    //==========================================================
    // 21 — WAIT HOMING COMPLETE
    //==========================================================
    21:
        // Start infeed/outfeed only after homing is complete
//        IF lowerKnifeStatusW1.homingComplete THEN
            lowerKnifeInFeedRun  := TRUE;
            lowerKnifeOutFeedRun := TRUE;
            lowerKnifeStep := 40;
//        END_IF

    //==========================================================
    // 40 — NORMAL OPERATION
    //==========================================================
    40:
	
        lowerKnifeJogFw       := lowerKnifeJogFwCmd;
        lowerKnifeJogRev      := lowerKnifeJogRevCmd;	
	
		instTOF_LowerKnifePaperSensor(IN := lowerKnifePaperSensor, PT:= T#30M);	
	
		IF instTOF_LowerKnifePaperSensor.Q  OR lineSpeedMPM > 5 THEN
			
			lowerKnifeInFeedDriveRef := LIMIT(machineConfigLowerKnife.minLineSpeed,
											  lineSpeedMPMRamp,
											  lowerLevelInfeedSpeedLimit) * machineConfigLowerKnife.infeedRollSpeedOffset;
		 
			lowerKnifeOutFeedDriveRef := LIMIT(machineConfigLowerKnife.minLineSpeed,
											   lineSpeedMPMRamp,
											   999) * machineConfigLowerKnife.outfeedRollSpeedOffset;		
		ELSE
			
			lowerKnifeInFeedDriveRef := 0;
			lowerKnifeOutFeedDriveRef := 0;		
			
		END_IF



        // Enable cut only when commanded and paper present
        lowerKnifeCut := (lowerKnifeCutCmd AND lowerKnifePaperSensor);
		
		
		IF NOT measuringWheelPaperPresence THEN
			
			lowerLevelInfeedSpeedLimit := lowerKnifeMaximumSpeedActive;
			
		ELSE
		
			lowerLevelInfeedSpeedLimit := 999;	
		
		END_IF				
		

END_CASE

//==============================================================
// 5) GLOBAL INTERLOCK — IMMEDIATE STOP
//==============================================================
// Immediate stop on any of these conditions:
// - Safety chain not OK
// - Any drive not OK
// - Power OFF command rising edge
IF (NOT safetyFeedback)
   OR (NOT lowerKnifeAllDrivesOK)
   OR lowerKnifeRtPowerOff.Q THEN

    lowerKnifeStep := 0;

    lowerKnifeEnable      := FALSE;
    lowerKnifeSlave1Run   := FALSE;
    lowerKnifeSlave2Run   := FALSE;
    lowerKnifeInFeedRun   := FALSE;
    lowerKnifeOutFeedRun  := FALSE;

    lowerKnifeJogFw       := FALSE;
    lowerKnifeJogRev      := FALSE;
    lowerKnifeHome        := FALSE;
    lowerKnifeCut         := FALSE;

    lowerKnifeInFeedDriveRef  := 0.0;
    lowerKnifeOutFeedDriveRef := 0.0;

    // Reset internal timers for a clean restart
    lowerKnifeTimerWait(IN := FALSE);
    lowerKnifeTimerPulse(IN := FALSE);
    lowerKnifeTimerClear(IN := FALSE);
    lowerKnifeTimerReset(IN := FALSE);
END_IF

//Start Lubrification pump
lowerKnifeLubrification := lowerKnifeEnable;
 


//==============================================================
// ENCODER SELECTION — LOWER KNIFE
//==============================================================
// Copied 1:1 from the provided upper-knife reference logic.
// NOTE: The TRUE/FALSE meaning of "*EncoderSwitch" should match your IO mapping.
//==============================================================


   //----------------------------------------------------------
    // AUTO MODE
    //----------------------------------------------------------
    IF NOT measuringWheelPaperPresence THEN
        // No paper → immediate fallback to measuring wheel encoder
        lowerKnifeEncoderSwitch := TRUE;

        // Reset delay timer
        instTONLowerKnifeSwitchEncoderDelay.IN := FALSE;

    ELSE
        // Paper present → start delay before switching
        instTONLowerKnifeSwitchEncoderDelay.IN := TRUE;

        // Switch only after delay elapsed
        IF instTONLowerKnifeSwitchEncoderDelay.Q THEN
				
			lowerKnifeEncoderSwitch := FALSE;

        END_IF
		
    END_IF

//--------------------------------------------------------------
// TIMER EXECUTION (ALWAYS CALLED)
//--------------------------------------------------------------
instTONLowerKnifeSwitchEncoderDelay(
    PT := machineConfigLowerKnife.switchEncoderDelay
);
END_METHOD

METHOD _03_LineSpeedLimit
VAR_INPUT
END_VAR
//==============================================================
// SHEET LENGTH SELECTION — UPPER / LOWER KNIFE
//==============================================================

CASE currentOrder.levelSelector OF

    //----------------------------------------------------------
    // ORDER 1 ONLY
    //----------------------------------------------------------
    E_LevelSelector.eUpperOnly:
         instFB_SpeedLimitUpperKnife.sheetLength := currentOrder.order1.sheetLength;
		instFB_SpeedLimitLowerKnife.sheetLength := currentOrder.order1.sheetLength;
	 
		instFB_SpeedLimitUpperKnife.knifeEnabled := TRUE;
		instFB_SpeedLimitLowerKnife.knifeEnabled := FALSE;	
    //----------------------------------------------------------
    // ORDER 2 ONLY
    //----------------------------------------------------------
    E_LevelSelector.eLowerOnly:
        instFB_SpeedLimitLowerKnife.sheetLength := currentOrder.order1.sheetLength;
			instFB_SpeedLimitLowerKnife.sheetLength := currentOrder.order1.sheetLength;
	
		instFB_SpeedLimitUpperKnife.knifeEnabled := FALSE;
		instFB_SpeedLimitLowerKnife.knifeEnabled := TRUE;		

    //----------------------------------------------------------
    // BOTH ORDERS
    //----------------------------------------------------------
    E_LevelSelector.eBoth:

		// Inverted mapping
		instFB_SpeedLimitUpperKnife.sheetLength := currentOrder.order1.sheetLength;
		instFB_SpeedLimitLowerKnife.sheetLength := currentOrder.order2.sheetLength;
		instFB_SpeedLimitUpperKnife.knifeEnabled := TRUE;
		instFB_SpeedLimitLowerKnife.knifeEnabled := TRUE;
		

END_CASE

//==============================================================
// UPPER KNIFE — SPEED LIMIT CALCULATION
//==============================================================
instFB_SpeedLimitUpperKnife(
    machineSpeed             := lineSpeedMPM,
    numberOfPoints           := 10,
    machineConfigRotaryKnife := machineConfigUpperKnife,

    reduceLineSpeed          => upperKnifeReduceLineSpeed,
    speedLimitAcive          => upperKnifeSpeedLimit,
    speedCurveActive         => upperKnifeSpeedCurveActive,
    maximumSpeedActive       => upperKnifeMaximumSpeedActive
);

//==============================================================
// LOWER KNIFE — SPEED LIMIT CALCULATION
//==============================================================
instFB_SpeedLimitLowerKnife(
    machineSpeed             := lineSpeedMPM,
    numberOfPoints           := 10,
    machineConfigRotaryKnife := machineConfigLowerKnife,

    reduceLineSpeed          => lowerKnifeReduceLineSpeed,
    speedLimitAcive          => lowerKnifeSpeedLimit,
    speedCurveActive         => lowerKnifeSpeedCurveActive,
    maximumSpeedActive       => lowerKnifeMaximumSpeedActive
);
END_METHOD

METHOD _04_AuxControls
VAR_INPUT
END_VAR

//Start outfeed conveyor
startOutfeedConveyor := upperKnifeEnable OR lowerKnifeEnable;
END_METHOD

METHOD _05_DisplayVariables
VAR_INPUT
END_VAR
(*

    upperKnifeHmiStatus                       : hmiStatus_TypeStruct;
    lowerKnifeHmiStatus                       : hmiStatus_TypeStruct;

    reduceLineSpeed          => upperKnifeReduceLineSpeed,
    speedLimitAcive          => upperKnifeSpeedLimit,
    speedCurveActive         => upperKnifeSpeedCurveActive,
    maximumSpeedActive       => upperKnifeMaximumSpeedActive
	
    upperKnifeStatusW1              : rotaryKnifeStatusWord1_TypeStruct;
    upperKnifeStatusW2              : rotaryKnifeStatusWord2_TypeStruct;
rotaryKnifeStatusWord1_TypeStruct
rotaryKnifeStatusWord1_TypeStruct
    lowerKnifeStatusWord1           : INT;
    lowerKnifeStatusWord2           : INT;
    lowerKnifeModbusDword           : DWORD;
    lowerKnifeWriteMenu2029         : DWORD;
    lowerKnifeLineSpeed             : WORD;
    lowerKnifeStatusW1              : rotaryKnifeStatusWord1_TypeStruct;
    lowerKnifeStatusW2              : rotaryKnifeStatusWord2_TypeStruct;	
	
	
*)
//────────────────────────────────────────────
// LINE SPEED PROCESSING
//────────────────────────────────────────────
IF lineSpeedMPM > 0 THEN
    lineSpeed := TRUNC(lineSpeedMPM);
ELSE
    lineSpeed := 0;
END_IF

//────────────────────────────────────────────
// UPPER KNIFE - STATUS MAPPING
//────────────────────────────────────────────
upperKnifeHmiStatus.maxSpeed         := upperKnifeMaximumSpeedActive;       // Current active maximum speed
upperKnifeHmiStatus.speedLimitActive := upperKnifeSpeedLimit;                // Speed limit status
upperKnifeHmiStatus.speedCurveActive := upperKnifeSpeedCurveActive;

upperKnifeHmiStatus.statusWord1      := upperKnifeStatusW1;                 // General status word 1
upperKnifeHmiStatus.statusWord2      := upperKnifeStatusW2;                 // General status word 2
upperKnifeHmiStatus.totalOfCuts      := upperKnifeTotalOfCutsAccumulator;   // Cumulative cut counter
//────────────────────────────────────────────
// LOWER KNIFE - STATUS MAPPING
//────────────────────────────────────────────
lowerKnifeHmiStatus.maxSpeed         := lowerKnifeMaximumSpeedActive;       // Current active maximum speed
lowerKnifeHmiStatus.speedLimitActive := lowerKnifeSpeedLimit;                // Speed limit status
lowerKnifeHmiStatus.speedCurveActive := lowerKnifeSpeedCurveActive;

lowerKnifeHmiStatus.statusWord1      := lowerKnifeStatusW1;                 // General status word 1
lowerKnifeHmiStatus.statusWord2      := lowerKnifeStatusW2;                 // General status word 2
lowerKnifeHmiStatus.totalOfCuts      := lowerKnifeTotalOfCutsAccumulator;   // Cumulative cut counter
END_METHOD

METHOD _06_TotalOfCuts
VAR_INPUT
END_VAR
// ==========================================================
// UPPER KNIFE CUT DETECTION & COUNTER LOGIC
// ==========================================================

(* Detect rising edge of the upper knife sensor to increment the cut counter *)
IF upperKnifeHomeSensor AND NOT upperKnifeHomeSensorOld THEN
	
	// Increment the cumulative cut count for the upper knife
	upperKnifeTotalOfCutsAccumulator := upperKnifeTotalOfCutsAccumulator + 1;

END_IF

// Store current sensor state for next scan cycle edge detection
upperKnifeHomeSensorOld := upperKnifeHomeSensor;

(* Reset Logic: Clears the upper knife cut counter *)
IF upperKnifeReset THEN
	
	upperKnifeTotalOfCutsAccumulator := 0;

END_IF


// ==========================================================
// LOWER KNIFE CUT DETECTION & COUNTER LOGIC
// ==========================================================

(* Detect rising edge of the lower knife sensor to increment the cut counter *)
IF lowerKnifeHomeSensor AND NOT lowerKnifeHomeSensorOld THEN
	
	// Increment the cumulative cut count for the lower knife
	lowerKnifeTotalOfCutsAccumulator := lowerKnifeTotalOfCutsAccumulator + 1;

END_IF

// Store current sensor state for next scan cycle edge detection
lowerKnifeHomeSensorOld := lowerKnifeHomeSensor;

(* Reset Logic: Clears the lower knife cut counter *)
IF lowerKnifeReset THEN
	
	lowerKnifeTotalOfCutsAccumulator := 0;

END_IF
END_METHOD

METHOD _07_LineSpeedRamp
VAR
	
	rampTargetMPM : REAL;

END_VAR
(*

    lineSpeedMPM                    : REAL;
    aocSpeedMPM                     : REAL;
*)
IF NOT aocRunning THEN
	
	rampTargetMPM := lineSpeedMPM;

ELSE
	
	rampTargetMPM := aocSpeedMPM;

END_IF



// Ramp function block execution
instFB_Gen_SRamp(
    X          := rampTargetMPM,
    A_UP       := 5,
    A_DN       := -5,
    VU_MAX     := 1000.0,
    VD_MAX     := -1000.0,
    LIMIT_HIGH := 350,
	Y => lineSpeedMPMRamp
);




lineSpeedStacker := upperKnifeInFeedDriveRef;
END_METHOD

METHOD _08_StopTheLineCommand
VAR_INPUT
END_VAR

// ======================================================================
// Fault definition (ONLY using the variables you approved)
// ======================================================================
//
// Safety / guards / exhaust
// - safetyFeedback must be TRUE
// - guards open => fault
// - exhaust state must be consistent (one of them TRUE)
//   * both TRUE  => contradictory => fault
//   * both FALSE => unknown state  => fault
//
// Knives
// - guard closed must be TRUE
// - oil low / jam => fault
// - all drives OK must be TRUE
// - paper sensors: only considered fault if line is running (lineSpeedMPM > cMinRunSpeedMPM)
//
// Home sensors: typically should be validated only during homing,
// but since you requested them as alarm variables, we treat them as
// "unexpectedly active while running" (adjust if you prefer a different rule).
// ======================================================================

faultDetected :=
    // -----------------------
    // Safety / Guards
    // -----------------------
    (NOT safetyFeedback)
    OR NOT exitGuardClosed
    OR NOT infeedGuardClosed

    // -----------------------
    // Exhaust feedback consistency
    // -----------------------
//    OR (exhaustPressurized AND exhaustDepressurized)         // impossible/contradictory
//    OR ((NOT exhaustPressurized) AND (NOT exhaustDepressurized)) // no valid state

    // -----------------------
    // Upper knife conditions
    // -----------------------
    OR (NOT upperKnifeGuardClosed)
    OR NOT upperKnifeOilLevelLow
    OR upperKnifeJamDetected
    OR (NOT upperKnifeInfeedDrvOK)
    OR (NOT upperKnifeOutfeedDrvOK)
    OR (NOT upperKnifeMainDrvOK)
    OR (NOT upperKnifeSlave1DrvOK)
    OR (NOT upperKnifeSlave2DrvOK)

    // -----------------------
    // Lower knife conditions
    // -----------------------
    OR (NOT lowerKnifeGuardClosed)
    OR NOT lowerKnifeOilLevelLow
    OR lowerKnifeJamDetected
    OR (NOT lowerKnifeInfeedDrvOK)
    OR (NOT lowerKnifeOutfeedDrvOK)
    OR (NOT lowerKnifeMainDrvOK)
    OR (NOT lowerKnifeSlave1DrvOK)
    OR (NOT lowerKnifeSlave2DrvOK);


// ======================================================================
// Rising edge on fault => generate a 2s stop pulse
// ======================================================================
instRtrigFault(CLK := faultDetected);
instTP_LineStop(IN := instRtrigFault.Q, PT := T#2S);

// Line stop command (2 seconds pulse)
lineStop := instTP_LineStop.Q;
END_METHOD

METHOD _09_MeasuringWheel
VAR_INPUT
END_VAR

//Measuring wheel up down control
instTONMeasuringWheelDelay(
IN := measuringWheelPaperPresence,
PT := T#5S,
Q => measuringWheelSolenoid
);
END_METHOD

END_FUNCTION_BLOCK

// ---- Library/Ramp/FB_Gen_SRamp.TcPOU
FUNCTION_BLOCK FB_Gen_SRamp
VAR_INPUT
	X : REAL;
	A_UP : REAL  := 1.0;
	A_DN :REAL  := -1.0;;
	VU_MAX : REAL := 1.0;
	VD_MAX : REAL := -1.0;
	LIMIT_HIGH : REAL := 100.0;
	LIMIT_LOW : REAL := -100.0;
	RST : BOOL;
END_VAR
VAR_OUTPUT
	Y : REAL;
	V : REAL;
END_VAR
VAR
	cycle_time : TC_S;
	init: BOOL;
END_VAR

(* read the system_time in microseconds *)
cycle_time();

(* assure range of inputs *)
A_up := MAX(0.0, A_UP);
A_dn := MIN(0.0, A_dn);
VU_max := MAX(0.0, VU_max);
VD_max := MIN(0.0, VD_MAX);

(* calculate the output offset *)
IF rst OR NOT init THEN
	init := TRUE;
	Y := 0.0;
	V := 0.0;
ELSIF X = Y THEN
	v := 0.0;
ELSIF X > Y THEN
	(* output is too low >> ramp up and brake at the end *)
	(* accelerate the speed and limit to vu_max *)
	v := MIN(v + A_UP * cycle_time.TC, vu_max);
	(* calculate the max speed to be able to brake and select the lowest *)
	v := MIN(SQRT((Y-X) * 2.0 * A_DN), v);
	(* calculate the output and obey limits *)
	y := LIMIT(limit_low, y + MIN(v * cycle_time.TC, X-Y), limit_high);
ELSIF X < Y THEN
	(* output is too high >> ramp dn and brake at the end *)
	(* accelerate the speed and limit to vd_max *)
	v := MAX(v + A_DN * cycle_time.TC, vd_max);
	(* calculate the max speed to be able to brake and select the lowest *)
	v := MAX(-SQRT((Y-X) * 2.0 * A_UP), v);
	(* calculate the output and obey limits *)
	y := LIMIT(limit_low, y + MAX(v * cycle_time.TC, X-Y), limit_high);
END_IF;


(* revision history
hm	13. mar. 2008	rev 1.0
	original version

hm	11. mar. 2009	rev 1.1
	real constants updated to new systax using dot																																																																																																																																																																																																																																																																																																																																																																																																																																																																																																																																																																																																																																																																																																																																																																																																																																																																																																																																																																																																																																																											

*)

END_FUNCTION_BLOCK

// ---- Library/Machine/Rotary knife/Function Block/FB_SpeedLimit.TcPOU
FUNCTION_BLOCK FB_SpeedLimit
VAR_INPUT
	
	knifeEnabled			: BOOL;
    machineSpeed            : REAL; // Current machine speed (MPM)
    sheetLength             : REAL; // Length of the sheet being processed (MM)
    numberOfPoints          : INT;  // Total number of data points in the speed curve
    machineConfigRotaryKnife	: rotaryKnifeConfig_TypeStruct; // Configuration data for the rotary knife
END_VAR

VAR_OUTPUT
	reduceLineSpeed         : BOOL; // Flag indicating whether line speed should be reduced
	speedLimitAcive			: BOOL;
    speedCurveActive        : INT;  // Index of the active speed curve segment
	maximumSpeedActive		: REAL;	// Maximum speed for the current length
END_VAR

VAR
    index: INT; // Loop index
	count: DINT;
	nextPoint: INT;
	instGenPulse: GEN_PULSE;
END_VAR

// Ensure pulse generator is updated every scan
instGenPulse(ENQ:=TRUE, PTH:=T#100MS, PTL:=T#500MS);

IF knifeEnabled THEN
    // Reset status before checking
    reduceLineSpeed := FALSE;
    speedLimitAcive := FALSE;

    FOR index := 1 TO (numberOfPoints - 1) BY 1 DO
        nextPoint := index + 1;
        
        // Check if sheetLength falls within the current segment of the speed curve
        IF sheetLength >= machineConfigRotaryKnife.speedCurve[index].sheetLength AND 
           sheetLength < machineConfigRotaryKnife.speedCurve[nextPoint].sheetLength THEN
            
            // Reference the specific config for the current index to improve readability
            maximumSpeedActive := machineConfigRotaryKnife.speedCurve[index].machineSpeed;
            speedCurveActive := index;

            // Logic for speed reduction and warnings
            IF machineSpeed > maximumSpeedActive THEN
                reduceLineSpeed := instGenPulse.Q;
            END_IF
            
            // Warning threshold (5 units below max)
            speedLimitAcive := machineSpeed > (maximumSpeedActive - 5);
            
            // Exit loop early once the matching range is found
            EXIT; 
        END_IF
    END_FOR;
ELSE    
    speedLimitAcive := FALSE;
    reduceLineSpeed := FALSE;
    maximumSpeedActive := 0;
END_IF

END_FUNCTION_BLOCK

// ---- Library/Machine/DryEnd/AutomaticOrderChange/FB_AutomaticOrderChange_V1.TcPOU
FUNCTION_BLOCK FB_AutomaticOrderChange_V1
VAR_INPUT
    // ==============================
    // CONTROL
    // ==============================
    enable                      : BOOL;
    executeAOC                  : BOOL;     // Start automatic order change (level trigger)

    // ==============================
    // SENSORS
    // ==============================
    rotaryShearCutSensor        : BOOL;     // Rotary shear cut sensor
    measuringWheelPaperSensor   : BOOL;     // Measuring wheel sensor
    slitterPaperPresenceSensor  : BOOL;     // Slitter paper presence
    rotaryKnifePaperSensor      : BOOL;     // Rotary knife paper presence

    // ==============================
    // PROCESS VALUES
    // ==============================
    lineSpeedMPM                : REAL;     // Line speed [m/min]
    configuration               : aocConfig_TypeStruct; // AOC configuration parameters
END_VAR

VAR_IN_OUT
    currentOrder                : Order_TypeStruct;     // Current order details
    nextOrder                   : Order_TypeStruct;     // Next order details
END_VAR

VAR_OUTPUT
    // ==============================
    // STATUS
    // ==============================
    error                       : BOOL;
    aocRunning                  : BOOL;
    aocTimeOut                  : BOOL;
    statusDisplay               : STRING;

	
	rotaryShearCutX1Timeout		: BOOL;
	measuringWheelClearTimeout	: BOOL;
	slitterClearTimeout			: BOOL;
	rotaryKnifeClarTimeout		: BOOL;
	
    // ==============================
    // MACHINE COMMANDS
    // ==============================
    referenceSwitch             : BOOL;     // Switch between double facer and AOC ramp reference
    doubleFacerSpeedUP          : BOOL;
    doubleFacerSpeedDown        : BOOL;

    // ==============================
    // TRIGGERS / PULSES
    // ==============================
    rotaryShearCutX1            : BOOL;
    executePositioning          : BOOL;
    topStackerDischarge         : BOOL;
    bottomStackerDischarge      : BOOL;

    // ==============================
    // SPEED REFERENCES
    // ==============================
    rotaryKnifeSpeedRef         : LREAL;
    slitterKnifeSpeedRef        : LREAL;
    slitterScorerSpeedRef       : REAL;
END_VAR

VAR
    // ==============================
    // STATE MACHINE
    // ==============================
    stateMachine                : WORD;

    // ==============================
    // EDGE / INTERNAL LATCHES
    // ==============================
    enableOld                   : BOOL;
    executeAOC_Old              : BOOL;
    rExecuteAOC                 : BOOL;      // rising edge of executeAOC

    // ==============================
    // REQUESTS (drive FB inputs)
    // ==============================
    reqTpRotaryShear            : BOOL;
    reqTpExecutePositioning     : BOOL;
    reqTpStackerTop             : BOOL;
    reqTpStackerBottom          : BOOL;

    reqTonSlitterDelay          : BOOL;
    reqTonStackerDelay          : BOOL;
    reqTonChangeSheetLength     : BOOL;

    // ==============================
    // FUNCTION BLOCK INSTANCES
    // ==============================
    tpRotaryShear               : TP;
    tpExecutePositioning        : TP;
    tpStackerTop                : TP;
    tpStackerBottom             : TP;

    tonSlitterPresenceDelay     : TON;
    tonStackerDischargeDelay    : TON;
    tonChangeSheetLength        : TON;

    tonAocTimeout               : TON;

    instFB_Gen_SRamp            : FB_Gen_SRamp;
    instGEN_PULSESpeedCtrl      : GEN_PULSE;

    lineSpeedMPMRamp            : REAL;

    // ==============================
    // INTERNAL (optional)
    // ==============================
    aocSpeedTarget              : REAL;      // target line speed during AOC (m/min)
	

    // ------------------------------
    // Timeout supervision (max times)
    // ------------------------------
    reqTonShearCutMax           : BOOL;
    reqTonMeasWheelClearMax     : BOOL;
    reqTonSlitterClearMax       : BOOL;
    reqTonRotaryKnifeClearMax   : BOOL;

    tonShearCutMax              : TON;
    tonMeasWheelClearMax        : TON;
    tonSlitterClearMax          : TON;
    tonRotaryKnifeClearMax      : TON;

    // ------------------------------
    // Error pulse management (2s)
    // ------------------------------
    faultCode                   : USINT;   // 0=none, 1=shear, 2=measwheel, 3=slitter, 4=rotaryknife
    reqTpFaultPulse             : BOOL;
    tpFaultPulse                : TP;	
	
END_VAR

VAR CONSTANT
    // ==============================
    // LIFE CYCLE
    // ==============================
    STATUS_NO_CALL                  : WORD := 16#7000;
    STATUS_FB_FIRST_CALL            : WORD := 16#7001;

    // ==============================
    // AOC STATES
    // ==============================
    STATUS_CHECK_CONDITIONS         : WORD := 16#8000;
    STATUS_SAVE_DF_SPEED            : WORD := 16#8001;
    STATUS_REDUCE_DF_SPEED          : WORD := 16#8002;

    STATUS_ROTARY_SHEAR_CUT_X1      : WORD := 16#8003;
    STATUS_WAIT_ROTARY_SHEAR_CUT_X1 : WORD := 16#8103;

    STATUS_INCREASE_DRYEND_SPEED    : WORD := 16#8004;
    STATUS_CHANGE_SLT_ORDER         : WORD := 16#8005;
    STATUS_CHANGE_RK_SHEET_LENGTH   : WORD := 16#8006;
    STATUS_STK_DISCHARGE            : WORD := 16#8007;

    STATUS_AOC_FINISHED             : WORD := 16#8010;
    STATUS_ERROR                : WORD := 16#8FFF;	
	
END_VAR

// =================================================================================================
// CPNTeck - Automação ind.
// (c)Copyright 2022 All Rights Reserved
// -------------------------------------------------------------------------------------------------
// Purpose: Automatic Order Change (AOC) sequence controller.
// Steps (high-level):
//   1) Check material presence
//   2) Reduce double facer speed down to AOC speed
//   3) Execute single cut (rotary shear X1)
//   4) Switch reference to AOC ramp and clear dry-end/slitter
//   5) Update slitter parameters from nextOrder
//   6) Change rotary knife sheet length (delay / clearance window)
//   7) Discharge stacker
//   8) Finish and reset
//
// Notes (important):
// - TP/TON instances are called once per scan at the end of the FB.
// - Requests (reqTp*/reqTon*) are set inside the state machine.
// - This avoids conflicting multi-calls to the same FB instance.
// =================================================================================================


// =================================================================================================
// 1) EDGE HANDLING / DISABLE RESET
// =================================================================================================
rExecuteAOC := executeAOC AND NOT executeAOC_Old;
executeAOC_Old := executeAOC;

// Falling edge of enable => hard reset (safe state)
IF (NOT enable) AND enableOld THEN
    // ---- outputs ----
    error := FALSE;
    aocRunning := FALSE;
    aocTimeOut := FALSE;
    statusDisplay := 'Not running...';

    referenceSwitch := FALSE;
    doubleFacerSpeedUP := FALSE;
    doubleFacerSpeedDown := FALSE;

    rotaryShearCutX1 := FALSE;
    executePositioning := FALSE;
    topStackerDischarge := FALSE;
    bottomStackerDischarge := FALSE;

    rotaryKnifeSpeedRef := 0.0;
    slitterKnifeSpeedRef := 0.0;
    slitterScorerSpeedRef := 0.0;

    // ---- fault outputs ----
    rotaryShearCutX1Timeout := FALSE;
    measuringWheelClearTimeout := FALSE;
    slitterClearTimeout := FALSE;
    rotaryKnifeClarTimeout := FALSE;

    // ---- state ----
    stateMachine := STATUS_NO_CALL;

    // ---- reset requests ----
    reqTpRotaryShear := FALSE;
    reqTpExecutePositioning := FALSE;
    reqTpStackerTop := FALSE;
    reqTpStackerBottom := FALSE;

    reqTonSlitterDelay := FALSE;
    reqTonStackerDelay := FALSE;
    reqTonChangeSheetLength := FALSE;

    reqTonShearCutMax := FALSE;
    reqTonMeasWheelClearMax := FALSE;
    reqTonSlitterClearMax := FALSE;
    reqTonRotaryKnifeClearMax := FALSE;

    // ---- stop timeout ----
    tonAocTimeout.IN := FALSE;

    // ---- error pulse ----
    faultCode := 0;
    reqTpFaultPulse := FALSE;

    enableOld := enable;
    RETURN;
END_IF

// Rising edge of enable => initialize
IF enable AND (NOT enableOld) THEN
    stateMachine := STATUS_FB_FIRST_CALL;

    // Keep outputs in safe defaults
    error := FALSE;
    aocRunning := FALSE;
    aocTimeOut := FALSE;
    statusDisplay := 'Initialized';

    // fault outputs default
    rotaryShearCutX1Timeout := FALSE;
    measuringWheelClearTimeout := FALSE;
    slitterClearTimeout := FALSE;
    rotaryKnifeClarTimeout := FALSE;

    faultCode := 0;
    reqTpFaultPulse := FALSE;

    enableOld := enable;
    RETURN;
END_IF

// If not enabled, do nothing
IF NOT enable THEN
    enableOld := enable;
    RETURN;
END_IF

enableOld := enable;


// =================================================================================================
// 2) DEFAULTS EACH SCAN (avoid latching unwanted outputs)
// =================================================================================================
rotaryShearCutX1 := FALSE;
executePositioning := FALSE;
topStackerDischarge := FALSE;
bottomStackerDischarge := FALSE;

doubleFacerSpeedUP := FALSE;
doubleFacerSpeedDown := FALSE;

// Fault outputs: pulse-managed in STATUS_ERROR only
rotaryShearCutX1Timeout := FALSE;
measuringWheelClearTimeout := FALSE;
slitterClearTimeout := FALSE;
rotaryKnifeClarTimeout := FALSE;

// Requests default OFF; states will enable them as needed
reqTpRotaryShear := FALSE;
reqTpExecutePositioning := FALSE;
reqTpStackerTop := FALSE;
reqTpStackerBottom := FALSE;

reqTonSlitterDelay := FALSE;
reqTonStackerDelay := FALSE;
reqTonChangeSheetLength := FALSE;

// timeout requests
reqTonShearCutMax := FALSE;
reqTonMeasWheelClearMax := FALSE;
reqTonSlitterClearMax := FALSE;
reqTonRotaryKnifeClearMax := FALSE;

// error pulse request
reqTpFaultPulse := FALSE;


// =================================================================================================
// 3) TRIGGER AOC (rising edge)
// =================================================================================================
IF rExecuteAOC THEN
    aocTimeOut := FALSE;
    faultCode := 0;
    stateMachine := STATUS_CHECK_CONDITIONS;
END_IF


// =================================================================================================
// 4) STATE MACHINE
// =================================================================================================
CASE stateMachine OF

    STATUS_FB_FIRST_CALL:
        statusDisplay := 'FB first call';
        stateMachine := STATUS_NO_CALL;

    STATUS_NO_CALL:
        statusDisplay := 'Idle';
        aocRunning := FALSE;
        referenceSwitch := FALSE;
        tonAocTimeout.IN := FALSE;
        faultCode := 0;
		//Write the line speed
        instFB_Gen_SRamp.X          := lineSpeedMPM;
        instFB_Gen_SRamp.LIMIT_LOW  := lineSpeedMPM;     // don’t ramp below current
        instFB_Gen_SRamp.LIMIT_HIGH := lineSpeedMPM;		
		

    STATUS_CHECK_CONDITIONS:
        statusDisplay := 'Checking conditions';

        // Must have paper present everywhere to proceed
        IF (NOT measuringWheelPaperSensor)
           OR (NOT slitterPaperPresenceSensor)
           OR (NOT rotaryKnifePaperSensor) THEN

            // Not safe to run AOC, finish immediately
            stateMachine := STATUS_AOC_FINISHED;
        ELSE
            // Start timeout supervision (global AOC timeout)
            tonAocTimeout.IN := TRUE;
            tonAocTimeout.PT := configuration.aocTimeout;

            stateMachine := STATUS_SAVE_DF_SPEED;
        END_IF


    STATUS_SAVE_DF_SPEED:
        statusDisplay := 'STATUS_SAVE_DF_SPEED';
        aocRunning := TRUE;

        // Compute AOC target speed (m/min)
        aocSpeedTarget := configuration.automaticOrderChangeSpeed * configuration.automaticOrderChangeSpeedMult;

        stateMachine := STATUS_REDUCE_DF_SPEED;


    STATUS_REDUCE_DF_SPEED:
        statusDisplay := 'STATUS_REDUCE_DF_SPEED';

        // While above AOC speed => pulse DF speed down
        IF lineSpeedMPM > configuration.automaticOrderChangeSpeed THEN
            doubleFacerSpeedDown := instGEN_PULSESpeedCtrl.Q;
        ELSE
            // Reached speed => go cut
            stateMachine := STATUS_ROTARY_SHEAR_CUT_X1;
        END_IF

        // Freeze ramp output to current speed (no AOC ramp yet)
        instFB_Gen_SRamp.X          := lineSpeedMPM;
        instFB_Gen_SRamp.LIMIT_LOW  := lineSpeedMPM;
        instFB_Gen_SRamp.LIMIT_HIGH := lineSpeedMPM;


    STATUS_ROTARY_SHEAR_CUT_X1:
        statusDisplay := 'Cutting web (X1)';
        // Generate a 1s pulse to the shear output
        reqTpRotaryShear := TRUE;

        // Start max-time supervision for shear confirmation
        reqTonShearCutMax := TRUE;

        stateMachine := STATUS_WAIT_ROTARY_SHEAR_CUT_X1;


    STATUS_WAIT_ROTARY_SHEAR_CUT_X1:
        statusDisplay := 'Waiting shear sensor';

        // Keep supervising max time while waiting
        reqTonShearCutMax := TRUE;

        IF rotaryShearCutSensor THEN
            // Stop supervision timer
            reqTonShearCutMax := FALSE;

            // Switch reference to AOC ramp
            referenceSwitch := TRUE;
            stateMachine := STATUS_INCREASE_DRYEND_SPEED;

        ELSIF tonShearCutMax.Q THEN
            // Timeout => go error, pulse output 2s, then idle
            reqTonShearCutMax := FALSE;
            faultCode := 1; // shear timeout
            stateMachine := STATUS_ERROR;
        END_IF


    STATUS_INCREASE_DRYEND_SPEED:
        statusDisplay := 'Clearing dry-end / slitter';

        // Start max-time supervision while waiting for measuring wheel to clear
        reqTonMeasWheelClearMax := TRUE;

        // Wait until measuring wheel area clears
        IF NOT measuringWheelPaperSensor THEN
            reqTonMeasWheelClearMax := FALSE;
            stateMachine := STATUS_CHANGE_SLT_ORDER;

        ELSIF tonMeasWheelClearMax.Q THEN
            reqTonMeasWheelClearMax := FALSE;
            faultCode := 2; // measuring wheel clear timeout
            stateMachine := STATUS_ERROR;
        END_IF

        // Apply AOC speed ramp (raise limit high to target)
        instFB_Gen_SRamp.X          := aocSpeedTarget;
        instFB_Gen_SRamp.LIMIT_LOW  := lineSpeedMPM;     // don’t ramp below current
        instFB_Gen_SRamp.LIMIT_HIGH := aocSpeedTarget;


    STATUS_CHANGE_SLT_ORDER:
        statusDisplay := 'Changing slitter order (when clear)';

        // Start max-time supervision for "slitter clear + delay window"
        reqTonSlitterClearMax := TRUE;

        // Copy only the parameters that need to switch during AOC
        currentOrder.fluteType     := nextOrder.fluteType;
        currentOrder.levelSelector := nextOrder.levelSelector;

        currentOrder.order1.sheetType     := nextOrder.order1.sheetType;
        currentOrder.order1.sheetQuantity := nextOrder.order1.sheetQuantity;
        currentOrder.order1.sheetM1       := nextOrder.order1.sheetM1;
        currentOrder.order1.sheetM2       := nextOrder.order1.sheetM2;
        currentOrder.order1.sheetM3       := nextOrder.order1.sheetM3;
        currentOrder.order1.sheetM4       := nextOrder.order1.sheetM4;
        currentOrder.order1.sheetM5       := nextOrder.order1.sheetM5;

        currentOrder.order2.sheetType     := nextOrder.order2.sheetType;
        currentOrder.order2.sheetQuantity := nextOrder.order2.sheetQuantity;
        currentOrder.order2.sheetM1       := nextOrder.order2.sheetM1;
        currentOrder.order2.sheetM2       := nextOrder.order2.sheetM2;
        currentOrder.order2.sheetM3       := nextOrder.order2.sheetM3;
        currentOrder.order2.sheetM4       := nextOrder.order2.sheetM4;
        currentOrder.order2.sheetM5       := nextOrder.order2.sheetM5;

        // Start delay only after slitter area becomes clear
        IF NOT slitterPaperPresenceSensor THEN
            reqTonSlitterDelay := TRUE;
            tonSlitterPresenceDelay.PT := configuration.slitterPaperPresenceDelay;
        END_IF

        IF tonSlitterPresenceDelay.Q THEN
            // Success => stop max-time supervision
            reqTonSlitterClearMax := FALSE;

            // Pulse executePositioning
            reqTpExecutePositioning := TRUE;

            // stop delay timer (will reset by IN=FALSE)
            reqTonSlitterDelay := FALSE;

            stateMachine := STATUS_CHANGE_RK_SHEET_LENGTH;

        ELSIF tonSlitterClearMax.Q THEN
            // Timeout => error
            reqTonSlitterClearMax := FALSE;
            reqTonSlitterDelay := FALSE;
            faultCode := 3; // slitter clear timeout
            stateMachine := STATUS_ERROR;
        END_IF


    STATUS_CHANGE_RK_SHEET_LENGTH:
        statusDisplay := 'Changing rotary knife sheet length';

        // Start max-time supervision for rotary knife clear
        reqTonRotaryKnifeClearMax := TRUE;

        // Allow a clearance window for RK sheet length change (time-based + sensor-based)
        reqTonChangeSheetLength := TRUE;
        tonChangeSheetLength.PT := configuration.changeSheetLengthTime;

        // When RK is clear OR changeSheetLength window elapsed => proceed
        IF (NOT rotaryKnifePaperSensor) OR tonChangeSheetLength.Q THEN
            reqTonRotaryKnifeClearMax := FALSE;
            reqTonChangeSheetLength := FALSE;

            stateMachine := STATUS_STK_DISCHARGE;

        ELSIF tonRotaryKnifeClearMax.Q THEN
            // Timeout => error
            reqTonRotaryKnifeClearMax := FALSE;
            reqTonChangeSheetLength := FALSE;
            faultCode := 4; // rotary knife clear timeout
            stateMachine := STATUS_ERROR;
        END_IF


    STATUS_STK_DISCHARGE:
        statusDisplay := 'Discharging stacker';

        // Delay before discharge
        reqTonStackerDelay := TRUE;
        tonStackerDischargeDelay.PT := configuration.stackerDischargeDelay;

        IF tonStackerDischargeDelay.Q THEN
            // Pulse discharge commands
            currentOrder.changeOrderRequest := TRUE;

            reqTpStackerTop := TRUE;
            reqTpStackerBottom := TRUE;

            stateMachine := STATUS_AOC_FINISHED;
        END_IF


    STATUS_ERROR:
        // Error state: pulse the corresponding timeout output for 2 seconds, then go Idle (NO_CALL)
        aocRunning := FALSE;
        referenceSwitch := FALSE;
        doubleFacerSpeedUP := FALSE;
        doubleFacerSpeedDown := FALSE;

        // Stop AOC timeout supervision
        tonAocTimeout.IN := FALSE;

        // Request 2s fault pulse
        reqTpFaultPulse := TRUE;

        CASE faultCode OF
            1: statusDisplay := 'ERROR: rotaryShearCutX1 timeout';
            2: statusDisplay := 'ERROR: measuringWheel clear timeout';
            3: statusDisplay := 'ERROR: slitter clear timeout';
            4: statusDisplay := 'ERROR: rotaryKnife clear timeout';
        ELSE
            statusDisplay := 'ERROR: unknown';
        END_CASE

        // After pulse ends, return to idle (no reset required)
        IF NOT tpFaultPulse.Q THEN
            // tpFaultPulse.Q will go TRUE only after call; so this "end" check must be done with tpFaultPulse.IN logic:
            // We handle it by checking tpFaultPulse.Q and tpFaultPulse.IN in the FB call section below via tpFaultPulse output.
        END_IF
        // NOTE: actual transition to Idle is handled below after TP call (see section 7)


    STATUS_AOC_FINISHED:
        statusDisplay := 'AOC Finished';

        aocRunning := FALSE;
        referenceSwitch := FALSE;
        doubleFacerSpeedUP := FALSE;
        doubleFacerSpeedDown := FALSE;

        // Stop timeout monitoring
        tonAocTimeout.IN := FALSE;

        // Return to idle
        stateMachine := STATUS_NO_CALL;

END_CASE


// =================================================================================================
// 5) GLOBAL FUNCTION BLOCK CALLS (call once per scan)
// =================================================================================================

// Pulse generator for DF speed up/down buttons
instGEN_PULSESpeedCtrl(
    ENQ := TRUE,
    PTH := configuration.speedControlPulseONTime,
    PTL := configuration.speedControlPulseOFFTime
);

// Ramp block (driven by instFB_Gen_SRamp.X and limits set in states)
instFB_Gen_SRamp(
    A_UP    := configuration.rampUpTimeSec,
    A_DN    := configuration.rampDownTimeSec,
    VU_MAX  := 1000.0,
    VD_MAX  := -1000.0,
    Y       => lineSpeedMPMRamp
);

// Timers (existing)
tonSlitterPresenceDelay(IN := reqTonSlitterDelay);
tonStackerDischargeDelay(IN := reqTonStackerDelay);
tonChangeSheetLength(IN := reqTonChangeSheetLength);

tonAocTimeout(IN := tonAocTimeout.IN, PT := configuration.aocTimeout);

// Timers (new max-time supervision)
tonShearCutMax(IN := reqTonShearCutMax, PT := configuration.rotaryShearCutX1MaxTime);
tonMeasWheelClearMax(IN := reqTonMeasWheelClearMax, PT := configuration.measuringWheelClearMaxTime);
tonSlitterClearMax(IN := reqTonSlitterClearMax, PT := configuration.slitterClearMaxTime);
tonRotaryKnifeClearMax(IN := reqTonRotaryKnifeClearMax, PT := configuration.rotaryKnifeClearMaxTime);

// Pulses (existing)
tpRotaryShear(IN := reqTpRotaryShear, PT := T#1S, Q => rotaryShearCutX1);
tpExecutePositioning(IN := reqTpExecutePositioning, PT := T#1S, Q => executePositioning);
tpStackerTop(IN := reqTpStackerTop, PT := T#1S, Q => topStackerDischarge);
tpStackerBottom(IN := reqTpStackerBottom, PT := T#1S, Q => bottomStackerDischarge);

// Fault pulse (new)
tpFaultPulse(IN := reqTpFaultPulse, PT := T#2S);


// =================================================================================================
// 6) REFERENCES (derived from ramp output)
// =================================================================================================
rotaryKnifeSpeedRef   := lineSpeedMPMRamp * configuration.rotaryKnifeSpeedMult;
slitterKnifeSpeedRef  := lineSpeedMPMRamp * configuration.slitterSpeedMult;
slitterScorerSpeedRef := lineSpeedMPMRamp * configuration.slitterSpeedMult;


// =================================================================================================
// 7) ERROR OUTPUT PULSE + AUTO-RETURN TO IDLE (no reset required)
// =================================================================================================
IF stateMachine = STATUS_ERROR THEN
    // Pulse the selected fault output for 2s
    CASE faultCode OF
        1: rotaryShearCutX1Timeout := tpFaultPulse.Q;
        2: measuringWheelClearTimeout := tpFaultPulse.Q;
        3: slitterClearTimeout := tpFaultPulse.Q;
        4: rotaryKnifeClarTimeout := tpFaultPulse.Q;
    END_CASE

    // When TP finishes, return to idle
    IF (NOT tpFaultPulse.Q) AND (NOT reqTpFaultPulse) THEN
        // no action
    END_IF

    // Better end condition: TP done when IN went TRUE and Q returned FALSE.
    // We detect end by: reqTpFaultPulse is TRUE only inside STATUS_ERROR,
    // so after first scan it stays TRUE; we must drop it once TP is running.
    // Do that here:
    reqTpFaultPulse := FALSE;

    // Once TP has finished (Q=FALSE after being TRUE), go idle.
    // Easiest: if TP is not active anymore and we already dropped IN:
    IF (NOT tpFaultPulse.Q) THEN
        faultCode := 0;
        stateMachine := STATUS_NO_CALL;
    END_IF
END_IF


// =================================================================================================
// 8) TIMEOUT HANDLING (global AOC timeout)
// =================================================================================================
IF tonAocTimeout.Q THEN
    tonAocTimeout.IN := FALSE;
    aocTimeOut := TRUE;
    stateMachine := STATUS_AOC_FINISHED;
END_IF

END_FUNCTION_BLOCK

// ---- Library/Machine/DryEnd/Alarm Control/FB_AlarmControl.TcPOU
FUNCTION_BLOCK FB_AlarmControl
VAR_INPUT
    reset                           : BOOL; // Reset alarms command
    
    // General Faults
    safetyCircuitFault              : BOOL; // Alarm active - Safety circuit fault
    slitterHomeNotCompleteFault     : BOOL; // Alarm active - Slitter homing not complete
    slitterTractionNotEnabledFault  : BOOL; // Alarm active - Slitter traction not enabled
    
    // Knife Faults
    knife01Fault                    : BOOL; // Alarm active - Knife 01 fault
    knife02Fault                    : BOOL; // Alarm active - Knife 02 fault
    knife03Fault                    : BOOL; // Alarm active - Knife 03 fault
    knife04Fault                    : BOOL; // Alarm active - Knife 04 fault
    knife05Fault                    : BOOL; // Alarm active - Knife 05 fault
    knife06Fault                    : BOOL; // Alarm active - Knife 06 fault
    knife07Fault                    : BOOL; // Alarm active - Knife 07 fault
    
    // Upper Scorer Faults
    upperScorer01Fault              : BOOL; // Alarm active - Upper Scorer 01 fault
    upperScorer02Fault              : BOOL; // Alarm active - Upper Scorer 02 fault
    upperScorer03Fault              : BOOL; // Alarm active - Upper Scorer 03 fault
    upperScorer04Fault              : BOOL; // Alarm active - Upper Scorer 04 fault
    upperScorer05Fault              : BOOL; // Alarm active - Upper Scorer 05 fault
    upperScorer06Fault              : BOOL; // Alarm active - Upper Scorer 06 fault
    upperScorer07Fault              : BOOL; // Alarm active - Upper Scorer 07 fault
    upperScorer08Fault              : BOOL; // Alarm active - Upper Scorer 08 fault
    upperScorer09Fault              : BOOL; // Alarm active - Upper Scorer 09 fault
    upperScorer10Fault              : BOOL; // Alarm active - Upper Scorer 10 fault
    upperScorer11Fault              : BOOL; // Alarm active - Upper Scorer 11 fault
    upperScorer12Fault              : BOOL; // Alarm active - Upper Scorer 12 fault
    
    // Lower Scorer Faults
    lowerScorer01Fault              : BOOL; // Alarm active - Lower Scorer 01 fault
    lowerScorer02Fault              : BOOL; // Alarm active - Lower Scorer 02 fault
    lowerScorer03Fault              : BOOL; // Alarm active - Lower Scorer 03 fault
    lowerScorer04Fault              : BOOL; // Alarm active - Lower Scorer 04 fault
    lowerScorer05Fault              : BOOL; // Alarm active - Lower Scorer 05 fault
    lowerScorer06Fault              : BOOL; // Alarm active - Lower Scorer 06 fault
    lowerScorer07Fault              : BOOL; // Alarm active - Lower Scorer 07 fault
    lowerScorer08Fault              : BOOL; // Alarm active - Lower Scorer 08 fault
    lowerScorer09Fault              : BOOL; // Alarm active - Lower Scorer 09 fault
    lowerScorer10Fault              : BOOL; // Alarm active - Lower Scorer 10 fault
    lowerScorer11Fault              : BOOL; // Alarm active - Lower Scorer 11 fault
    lowerScorer12Fault              : BOOL; // Alarm active - Lower Scorer 12 fault

    // Traction and Axis Faults
    scorerTractionFault             : BOOL; // Alarm active - Scorer traction fault
    knifeTractionFault              : BOOL; // Alarm active - Knife traction fault
    scorerHeightAxisFault           : BOOL; // Alarm active - Scorer height axis fault
    scrapTrimOperatorSideFault      : BOOL; // Alarm active - Scrap trim operator side fault
    scrapTrimDriveSideFault         : BOOL; // Alarm active - Scrap trim drive side fault
    
    // Rotary Knife Specific Alarms
    exitGuardOpen                   : BOOL; // Alarm active - Exit guard open
    infeedGuardOpen                 : BOOL; // Alarm active - Infeed guard open
    exhaustDepressurized            : BOOL; // Alarm active - Exhaust system depressurized
    upperKnifeGuardClosed           : BOOL; // Alarm active - Upper knife guard open (Low Active)
    upperKnifeOilLevelLow           : BOOL; // Alarm active - Upper knife oil level low
    upperKnifeJamDetected           : BOOL; // Alarm active - Upper knife jam detected
    upperKnifeInfeedDrvOK           : BOOL; // Alarm active - Upper knife infeed drive fault (Low Active)
    upperKnifeOutfeedDrvOK          : BOOL; // Alarm active - Upper knife outfeed drive fault (Low Active)
    upperKnifeMainDrvOK             : BOOL; // Alarm active - Upper knife main drive fault (Low Active)
    upperKnifeSlave1DrvOK           : BOOL; // Alarm active - Upper knife slave 1 drive fault (Low Active)
    upperKnifeSlave2DrvOK           : BOOL; // Alarm active - Upper knife slave 2 drive fault (Low Active)
	upperKnifeNotActive				: BOOL;
	upperKnifeCutDisabled			: BOOL;

    
	lowerKnifeGuardClosed           : BOOL; // Alarm active - Lower knife guard open (Low Active)
    lowerKnifeOilLevelLow           : BOOL; // Alarm active - Lower knife oil level low
    lowerKnifeJamDetected           : BOOL; // Alarm active - Lower knife jam detected
    lowerKnifeInfeedDrvOK           : BOOL; // Alarm active - Lower knife infeed drive fault (Low Active)
    lowerKnifeOutfeedDrvOK          : BOOL; // Alarm active - Lower knife outfeed drive fault (Low Active)
    lowerKnifeMainDrvOK             : BOOL; // Alarm active - Lower knife main drive fault (Low Active)
    lowerKnifeSlave1DrvOK           : BOOL; // Alarm active - Lower knife slave 1 drive fault (Low Active)
    lowerKnifeSlave2DrvOK           : BOOL; // Alarm active - Lower knife slave 2 drive fault (Low Active)
	lowerKnifeNotActive				: BOOL;
	lowerKnifeCutDisabled			: BOOL;
	
	
	orderFault			:BOOL;

	knife1OutOfRange	:BOOL;
	knife2OutOfRange	:BOOL;
	knife3OutOfRange	:BOOL;
	knife4OutOfRange	:BOOL;
	knife5OutOfRange	:BOOL;
	
	scorer1OutOfRange	:BOOL;
	scorer2OutOfRange	:BOOL;
	scorer3OutOfRange	:BOOL;
	scorer4OutOfRange	:BOOL;
	scorer5OutOfRange	:BOOL;
	scorer6OutOfRange	:BOOL;
	scorer7OutOfRange	:BOOL;
	scorer8OutOfRange	:BOOL;
		
END_VAR

VAR_OUTPUT
    alarmsDisplay                   : hmiAlarms_TypeStruct; // Struct for HMI visualization
    alarmIndication                 : BOOL;                 // Global alarm active indicator
END_VAR

VAR
    alarmsVariables                 : hmiAlarms_TypeStruct; // Internal alarm latches
    resetOld                        : BOOL;                 // Rising edge detection for reset
END_VAR

_00_Reset();
_01_DryEnd();
_02_Slitter();
_03_RotaryKnife();
_08_AlarmIndication();

METHOD _00_Reset
VAR_INPUT
END_VAR
IF reset AND NOT resetOld THEN
	
	//Copy values from a holder variable with zero value to reset
	alarmsDisplay := alarmsVariables;
	
END_IF
END_METHOD

METHOD _01_DryEnd
VAR_INPUT
END_VAR


IF safetyCircuitFault THEN alarmsDisplay.slitter.safetyCircuitFault := safetyCircuitFault; END_IF
END_METHOD

METHOD _02_Slitter
VAR_INPUT
END_VAR
(*

	safetyCircuitFault							: BOOL;
	slitterHomeNotCompleteFault							: BOOL;
	slitterTractionNotEnabledFault					: BOOL;
*)




// ─────────────── KNIVES ───────────────
IF safetyCircuitFault THEN alarmsDisplay.slitter.knife01Fault := safetyCircuitFault; END_IF
IF slitterHomeNotCompleteFault THEN alarmsDisplay.slitter.slitterHomeNotCompleteFault := slitterHomeNotCompleteFault; END_IF
IF slitterTractionNotEnabledFault THEN alarmsDisplay.slitter.slitterTractionNotEnabledFault := slitterTractionNotEnabledFault; END_IF


// ─────────────── KNIVES ───────────────
IF knife01Fault THEN alarmsDisplay.slitter.knife01Fault := knife01Fault; END_IF
IF knife02Fault THEN alarmsDisplay.slitter.knife02Fault := knife02Fault; END_IF
IF knife03Fault THEN alarmsDisplay.slitter.knife03Fault := knife03Fault; END_IF
IF knife04Fault THEN alarmsDisplay.slitter.knife04Fault := knife04Fault; END_IF
IF knife05Fault THEN alarmsDisplay.slitter.knife05Fault := knife05Fault; END_IF
IF knife06Fault THEN alarmsDisplay.slitter.knife06Fault := knife06Fault; END_IF
IF knife07Fault THEN alarmsDisplay.slitter.knife07Fault := knife07Fault; END_IF

// ─────────────── SCORERS (UPPER) ───────────────
IF upperScorer01Fault THEN alarmsDisplay.slitter.upperScorer01Fault := upperScorer01Fault; END_IF
IF upperScorer02Fault THEN alarmsDisplay.slitter.upperScorer02Fault := upperScorer02Fault; END_IF
IF upperScorer03Fault THEN alarmsDisplay.slitter.upperScorer03Fault := upperScorer03Fault; END_IF
IF upperScorer04Fault THEN alarmsDisplay.slitter.upperScorer04Fault := upperScorer04Fault; END_IF
IF upperScorer05Fault THEN alarmsDisplay.slitter.upperScorer05Fault := upperScorer05Fault; END_IF
IF upperScorer06Fault THEN alarmsDisplay.slitter.upperScorer06Fault := upperScorer06Fault; END_IF
IF upperScorer07Fault THEN alarmsDisplay.slitter.upperScorer07Fault := upperScorer07Fault; END_IF
IF upperScorer08Fault THEN alarmsDisplay.slitter.upperScorer08Fault := upperScorer08Fault; END_IF
IF upperScorer09Fault THEN alarmsDisplay.slitter.upperScorer09Fault := upperScorer09Fault; END_IF
IF upperScorer10Fault THEN alarmsDisplay.slitter.upperScorer10Fault := upperScorer10Fault; END_IF
IF upperScorer11Fault THEN alarmsDisplay.slitter.upperScorer11Fault := upperScorer11Fault; END_IF
IF upperScorer12Fault THEN alarmsDisplay.slitter.upperScorer12Fault := upperScorer12Fault; END_IF

// ─────────────── SCORERS (LOWER) ───────────────
IF lowerScorer01Fault THEN alarmsDisplay.slitter.lowerScorer01Fault := lowerScorer01Fault; END_IF
IF lowerScorer02Fault THEN alarmsDisplay.slitter.lowerScorer02Fault := lowerScorer02Fault; END_IF
IF lowerScorer03Fault THEN alarmsDisplay.slitter.lowerScorer03Fault := lowerScorer03Fault; END_IF
IF lowerScorer04Fault THEN alarmsDisplay.slitter.lowerScorer04Fault := lowerScorer04Fault; END_IF
IF lowerScorer05Fault THEN alarmsDisplay.slitter.lowerScorer05Fault := lowerScorer05Fault; END_IF
IF lowerScorer06Fault THEN alarmsDisplay.slitter.lowerScorer06Fault := lowerScorer06Fault; END_IF
IF lowerScorer07Fault THEN alarmsDisplay.slitter.lowerScorer07Fault := lowerScorer07Fault; END_IF
IF lowerScorer08Fault THEN alarmsDisplay.slitter.lowerScorer08Fault := lowerScorer08Fault; END_IF
IF lowerScorer09Fault THEN alarmsDisplay.slitter.lowerScorer09Fault := lowerScorer09Fault; END_IF
IF lowerScorer10Fault THEN alarmsDisplay.slitter.lowerScorer10Fault := lowerScorer10Fault; END_IF
IF lowerScorer11Fault THEN alarmsDisplay.slitter.lowerScorer11Fault := lowerScorer11Fault; END_IF
IF lowerScorer12Fault THEN alarmsDisplay.slitter.lowerScorer12Fault := lowerScorer12Fault; END_IF

// ─────────────── ORDER / OUT OF RANGE ALARMS ───────────────
IF orderFault THEN alarmsDisplay.slitter.orderFault := orderFault; END_IF

// ─────────────── KNIVES OUT OF RANGE ───────────────
IF knife1OutOfRange THEN alarmsDisplay.slitter.knife1OutOfRange := knife1OutOfRange; END_IF
IF knife2OutOfRange THEN alarmsDisplay.slitter.knife2OutOfRange := knife2OutOfRange; END_IF
IF knife3OutOfRange THEN alarmsDisplay.slitter.knife3OutOfRange := knife3OutOfRange; END_IF
IF knife4OutOfRange THEN alarmsDisplay.slitter.knife4OutOfRange := knife4OutOfRange; END_IF
IF knife5OutOfRange THEN alarmsDisplay.slitter.knife5OutOfRange := knife5OutOfRange; END_IF

// ─────────────── SCORERS OUT OF RANGE ───────────────
IF scorer1OutOfRange THEN alarmsDisplay.slitter.scorer1OutOfRange := scorer1OutOfRange; END_IF
IF scorer2OutOfRange THEN alarmsDisplay.slitter.scorer2OutOfRange := scorer2OutOfRange; END_IF
IF scorer3OutOfRange THEN alarmsDisplay.slitter.scorer3OutOfRange := scorer3OutOfRange; END_IF
IF scorer4OutOfRange THEN alarmsDisplay.slitter.scorer4OutOfRange := scorer4OutOfRange; END_IF
IF scorer5OutOfRange THEN alarmsDisplay.slitter.scorer5OutOfRange := scorer5OutOfRange; END_IF
IF scorer6OutOfRange THEN alarmsDisplay.slitter.scorer6OutOfRange := scorer6OutOfRange; END_IF
IF scorer7OutOfRange THEN alarmsDisplay.slitter.scorer7OutOfRange := scorer7OutOfRange; END_IF
IF scorer8OutOfRange THEN alarmsDisplay.slitter.scorer8OutOfRange := scorer8OutOfRange; END_IF

// ─────────────── TRACTION / HEIGHT ───────────────
IF scorerTractionFault THEN
    alarmsDisplay.slitter.scorerTractionFault := scorerTractionFault;
END_IF

IF knifeTractionFault THEN
    alarmsDisplay.slitter.knifeTractionFault := knifeTractionFault;
END_IF

IF scorerHeightAxisFault THEN
    alarmsDisplay.slitter.scorerHeightAxisFault := scorerHeightAxisFault;
END_IF

// ─────────────── SCRAP TRIM ───────────────
IF scrapTrimOperatorSideFault THEN
    alarmsDisplay.slitter.scrapTrimOperatorSideFault := scrapTrimOperatorSideFault;
END_IF

IF scrapTrimDriveSideFault THEN
    alarmsDisplay.slitter.scrapTrimDriveSideFault := scrapTrimDriveSideFault;
END_IF
END_METHOD

METHOD _03_RotaryKnife
VAR_INPUT
END_VAR
//────────────────────────────────────────────
// SAFETY / GUARDS
//────────────────────────────────────────────
IF exitGuardOpen THEN alarmsDisplay.rotaryKnife.exitGuardOpen := exitGuardOpen; END_IF
IF infeedGuardOpen THEN alarmsDisplay.rotaryKnife.infeedGuardOpen := infeedGuardOpen; END_IF
IF exhaustDepressurized THEN alarmsDisplay.rotaryKnife.exhaustDepressurized := exhaustDepressurized; END_IF

//────────────────────────────────────────────
// UPPER KNIFE ALARMS
//────────────────────────────────────────────
IF upperKnifeGuardClosed THEN alarmsDisplay.rotaryKnife.upperKnifeGuardClosed := TRUE; END_IF
IF upperKnifeOilLevelLow THEN alarmsDisplay.rotaryKnife.upperKnifeOilLevelLow := TRUE; END_IF
IF upperKnifeJamDetected THEN alarmsDisplay.rotaryKnife.upperKnifeJamDetected := TRUE; END_IF
IF upperKnifeInfeedDrvOK THEN alarmsDisplay.rotaryKnife.upperKnifeInfeedDrvOK := TRUE; END_IF
IF upperKnifeOutfeedDrvOK THEN alarmsDisplay.rotaryKnife.upperKnifeOutfeedDrvOK := TRUE; END_IF
IF upperKnifeMainDrvOK THEN alarmsDisplay.rotaryKnife.upperKnifeMainDrvOK := TRUE; END_IF
IF upperKnifeSlave1DrvOK THEN alarmsDisplay.rotaryKnife.upperKnifeSlave1DrvOK := TRUE; END_IF
IF upperKnifeSlave2DrvOK THEN alarmsDisplay.rotaryKnife.upperKnifeSlave2DrvOK := TRUE; END_IF
IF upperKnifeNotActive THEN alarmsDisplay.rotaryKnife.upperKnifeNotActive := TRUE; END_IF
IF upperKnifeCutDisabled THEN alarmsDisplay.rotaryKnife.upperKnifeCutDisabled := TRUE; END_IF

//────────────────────────────────────────────
// LOWER KNIFE ALARMS
//────────────────────────────────────────────
IF lowerKnifeGuardClosed THEN alarmsDisplay.rotaryKnife.lowerKnifeGuardClosed := TRUE; END_IF
IF lowerKnifeOilLevelLow THEN alarmsDisplay.rotaryKnife.lowerKnifeOilLevelLow := TRUE; END_IF
IF lowerKnifeJamDetected THEN alarmsDisplay.rotaryKnife.lowerKnifeJamDetected := TRUE; END_IF
IF lowerKnifeInfeedDrvOK THEN alarmsDisplay.rotaryKnife.lowerKnifeInfeedDrvOK := TRUE; END_IF
IF lowerKnifeOutfeedDrvOK THEN alarmsDisplay.rotaryKnife.lowerKnifeOutfeedDrvOK := TRUE; END_IF
IF lowerKnifeMainDrvOK THEN alarmsDisplay.rotaryKnife.lowerKnifeMainDrvOK := TRUE; END_IF
IF lowerKnifeSlave1DrvOK THEN alarmsDisplay.rotaryKnife.lowerKnifeSlave1DrvOK := TRUE; END_IF
IF lowerKnifeSlave2DrvOK THEN alarmsDisplay.rotaryKnife.lowerKnifeSlave2DrvOK := TRUE; END_IF
IF lowerKnifeNotActive THEN alarmsDisplay.rotaryKnife.lowerKnifeNotActive := TRUE; END_IF
IF lowerKnifeCutDisabled THEN alarmsDisplay.rotaryKnife.lowerKnifeCutDisabled := TRUE; END_IF
END_METHOD

METHOD _08_AlarmIndication

VAR
	
	alarmCompResult	: DINT;

END_VAR

alarmCompResult := MEMCMP(pBuf1:= ADR(alarmsVariables) , pBuf2:= ADR(alarmsDisplay) , n:= SIZEOF(alarmsDisplay));

//alarmCompResult := alarmsVariables <> alarmsDisplay;

IF alarmCompResult <> 0 THEN

	alarmIndication := TRUE;
ELSE
	
	alarmIndication := FALSE;
	
END_IF
END_METHOD

END_FUNCTION_BLOCK

// ---- Library/Beckhoff/CX9020/FB_SavePersistentData.TcPOU
FUNCTION_BLOCK FB_SavePersistentData
VAR_INPUT
END_VAR
VAR_OUTPUT
END_VAR
VAR
	
	instFbClkPrgWritePersistentData: CLK_PRG;
	instFbWritePersistentData: FB_WritePersistentData;
	savePersisteData: BOOL;
	cpuPowerFailDetected: BOOL;
	writePersistentDataBusy: BOOL;
	writePersistentDataErr: BOOL;
	instFBSUpsBapi: FB_S_UPS_CX9020_U900;
	
	writePersistentDataErrId :UDINT;
END_VAR

VAR PERSISTENT
		
	saveCounter: DINT;

END_VAR
VAR // added by the converter: edge detectors and wires of the graphical bodies
    _w1 : DINT;
END_VAR

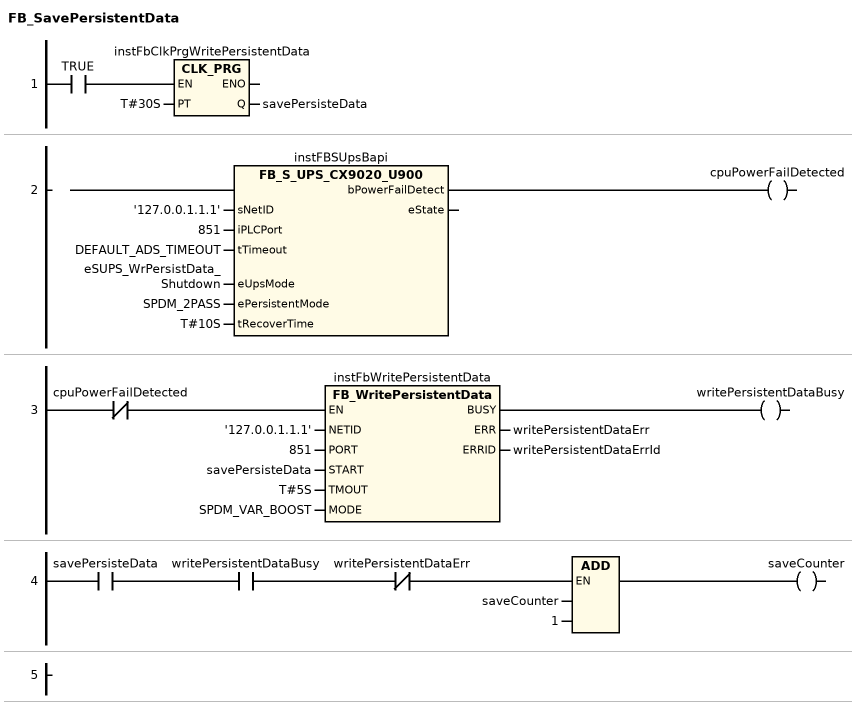
// NETWORK 1
instFbClkPrgWritePersistentData(PT := T#30S, Q => savePersisteData); // CLK_PRG

// NETWORK 2
instFBSUpsBapi(
    sNetID := '127.0.0.1.1.1',
    iPLCPort := 851,
    tTimeout := DEFAULT_ADS_TIMEOUT,
    eUpsMode := eSUPS_WrPersistData_Shutdown,
    ePersistentMode := SPDM_2PASS,
    tRecoverTime := T#10S); // FB_S_UPS_CX9020_U900
cpuPowerFailDetected := instFBSUpsBapi.bPowerFailDetect;

// NETWORK 3
IF NOT cpuPowerFailDetected THEN
    instFbWritePersistentData(
        NETID := '127.0.0.1.1.1',
        PORT := 851,
        START := savePersisteData,
        TMOUT := T#5S,
        MODE := SPDM_VAR_BOOST,
        ERR => writePersistentDataErr,
        ERRID => writePersistentDataErrId); // FB_WritePersistentData
END_IF
writePersistentDataBusy := instFbWritePersistentData.BUSY;

// NETWORK 4
IF savePersisteData AND writePersistentDataBusy AND NOT writePersistentDataErr THEN _w1 := saveCounter + 1; END_IF
saveCounter := _w1;

// NETWORK 5

END_FUNCTION_BLOCK

// ---- Library/Machine/Stacker/Simple/FB_SimpleSheetStackerControl.TcPOU
FUNCTION_BLOCK FB_SimpleSheetStackerControl
VAR_INPUT

    //==============================================================
    // Group command inputs
    //==============================================================
    startCmd                            : BOOL;
    stopCmd                             : BOOL;
    resetCmd                            : BOOL;


    //==============================================================
    // Speed reference inputs
    //==============================================================
    lineSpeedMPM                        : REAL;

    // EN: Current sheet length [mm].
    // PT: Comprimento atual da chapa [mm].
    sheetLengthMm                       : REAL;


    //==============================================================
    // Package command input
    //==============================================================
    // EN: Maintained automatic request. It is accepted once and remains
    //     blocked until the command returns to FALSE.
    // PT: Solicitação automática mantida. É aceita uma vez e permanece
    //     bloqueada até o comando retornar para FALSE.
    packageCompleteCmd                  : BOOL;

    // EN: Rising edge requests a complete discharge cycle for batch change.
    // PT: Borda de subida solicita um ciclo completo de descarte para troca de lote.
    changeBatchCmd                      : BOOL;

    // EN: Rising edge requests a local stack unload.
    // PT: Borda de subida solicita um descarte local da pilha.
    stackerUnloadCmd                    : BOOL;

	sheetConveyorsSpeedUpCmd : BOOL;

    //==============================================================
    // Machine configuration
    //==============================================================
    machineConfig                       : SimpleStackerConfig_TypeStruct;


    //==============================================================
    // Safety input
    //==============================================================
    safetyCircuitOk                     : BOOL;


    //==============================================================
    // Synchronized conveyor drive status inputs
    //==============================================================
    sheetConveyor1DriveOk               : BOOL;
    sheetConveyor2DriveOk               : BOOL;
    sheetConveyor3DriveOk               : BOOL;
    conveyorLevelerDriveOk              : BOOL;


    //==============================================================
    // Auxiliary drive status inputs
    //==============================================================
    backstopDriveOk                     : BOOL;

	//==============================================================
	// Sheet stack discharge conveyor drive status input
	//==============================================================
    sheetStackDischargeConveyorDriveOk                 : BOOL;

	
    //==============================================================
    // Position / measurement inputs
    //==============================================================
    stackHeightMm                       : REAL;
    backstopPositionMm                  : REAL;
    conveyorLevelerPositionMm           : REAL;


	//==============================================================
	// Conveyor leveler command inputs
	//==============================================================
	// EN: Starts conveyor leveler homing cycle.
	// PT: Inicia o ciclo de homing do nivelador da esteira.
	conveyorLevelerHomeCmd              : BOOL;
	
	// EN: Enables automatic leveling according to stack height.
	// PT: Habilita nivelamento automático conforme altura da pilha.
	conveyorLevelerAutoCmd              : BOOL;
	
	// EN: Manual up command.
	// PT: Comando manual para subir.
	conveyorLevelerUpCmd                : BOOL;
	
	// EN: Manual down command.
	// PT: Comando manual para descer.
	conveyorLevelerDownCmd              : BOOL;


    //==============================================================
    // Conveyor leveler limit inputs
    //==============================================================
    conveyorLevelerUpperSafetyLimit     : BOOL;
    conveyorLevelerLowerSafetyLimit     : BOOL;

    conveyorLevelerUpperLimit           : BOOL;
    conveyorLevelerLowerLimit           : BOOL;


    //==============================================================
    // Backstop command inputs
    //==============================================================
    // EN: Starts the backstop homing cycle.
    // PT: Inicia o ciclo de homing do backstop.
    backstopHomeCmd                     : BOOL;
	
    // EN: Starts the backstop homing cycle.
    // PT: Inicia o ciclo de homing do backstop.
    backstopExecutePositioningCmd			 : BOOL;
    // EN: Enables automatic positioning according to sheet length.
    // PT: Habilita posicionamento automático conforme comprimento da chapa.
    backstopAutoCmd                     : BOOL;

    // EN: Manual open command.
    // PT: Comando manual para abrir.
    backstopOpenCmd                     : BOOL;

    // EN: Manual close command.
    // PT: Comando manual para fechar.
    backstopCloseCmd                    : BOOL;


    //==============================================================
    // Backstop limit inputs
    //==============================================================
    backstopSafeMaxLimit                    : BOOL;	
    backstopMaxLimit                 	   	: BOOL;
    backstopMinLimit                   		: BOOL;
    backstopSafeMinLimit                    : BOOL;


    //==============================================================
    // Sheet handling command inputs
    //==============================================================
	// EN: Enables the sheet stack alignment brush.
	// PT: Habilita a vassoura de alinhamento da pilha de chapas.
	sheetStackAlignmentBrushEnableCmd        : BOOL;

	sheetStackDischargeConveyorManualRunCmd : BOOL;
    noCrushRollersDownCmd                 	: BOOL;

	safetyFeedBack1 	: BOOL;
	safetyFeedBack2 	: BOOL;
	safetyFeedBack3 	: BOOL;
	safetyFeedBack4 	: BOOL;
	safetyFeedBack5 	: BOOL;
	safetyFeedBack6 	: BOOL;
	safetyFeedBack7 	: BOOL;
	safetyFeedBack8 	: BOOL;	
	safetyFeedBack9 	: BOOL;	
	safetyFeedBack10 	: BOOL;		
		
	
END_VAR


VAR_OUTPUT

	hmiAlarms : hmiAlarmsSimpleStacker_TypeStruct;
	hmiStatus : hmiStatusSimpleStacker_TypeStruct;
	stackerRunning : BOOL;
	alarmActive	: BOOL;
	stopMachinePulse : BOOL;
	reset 	: BOOL;

	// EN: TRUE during an accepted unload sequence or while a stacker axis
	//     executes homing. Intended to command an external warning siren.
	// PT: TRUE durante uma sequência de descarte aceita ou enquanto um eixo
	//     do stacker executa homing. Destinada ao comando de uma sirene externa.
	stackerUnloadActive                 : BOOL;

	//==============================================================
	// EN: Stack unload handshake outputs
	// PT: Saídas de handshake do descarte da pilha
	//==============================================================
	// EN: One-scan pulse when a local unload request is accepted.
	//     It can be used to reset the external pile quantity in Metrics.
	// PT: Pulso de um ciclo quando um pedido local de descarte é aceito.
	//     Pode ser usado para resetar a quantidade externa da pilha no Metrics.
	stackerUnloadAccepted               : BOOL;

	// EN: 20 ms pulse to reset the external stack counter after any
	//     automatic or local unload request is accepted.
	// PT: Pulso de 20 ms para resetar o contador externo da pilha após
	//     qualquer pedido automático ou local de descarte ser aceito.
	externalCounterReset                : BOOL;

    //==============================================================
    // Synchronized conveyor drive outputs
    //==============================================================
    sheetConveyor1Run                   : BOOL;
    sheetConveyor2Run                   : BOOL;
    sheetConveyor3Run                   : BOOL;
	
	//==============================================================
	// Conveyor leveler drive outputs
	//==============================================================
	// EN: Conveyor leveler up run command.
	// PT: Comando para subir o nivelador da esteira.
	conveyorLevelerRunUp                : BOOL;
	
	// EN: Conveyor leveler down run command.
	// PT: Comando para descer o nivelador da esteira.
	conveyorLevelerRunDown              : BOOL;
	
	//==============================================================
	// Conveyor leveler magnetic brake output
	//==============================================================
	// EN: Magnetic brake release output. TRUE = brake released.
	// PT: Saída de liberação do freio magnético. TRUE = freio liberado.
	conveyorLevelerBrakeRelease         : BOOL;	

    //==============================================================
    // Backstop drive outputs
    //==============================================================
    // EN: Backstop forward run command. Positive/opening direction.
    // PT: Comando frente do backstop. Direção positiva/abrir.
    backstopRunFw                       : BOOL;

    // EN: Backstop reverse run command. Negative/closing direction.
    // PT: Comando reverso do backstop. Direção negativa/fechar.
    backstopRunRev                      : BOOL;

	//==============================================================
	// Sheet stack discharge conveyor outputs
	//==============================================================
	// EN: Sheet stack discharge conveyor run command.
	// PT: Comando de giro da esteira de descarga da pilha.
	sheetStackDischargeConveyorRun          : BOOL;




    //==============================================================
    // Synchronized conveyor speed reference outputs
    //==============================================================
    sheetConveyor1SpeedRefMPM           : REAL;
    sheetConveyor2SpeedRefMPM           : REAL;
    sheetConveyor3SpeedRefMPM           : REAL;
    conveyorLevelerSpeedRefMmps          : REAL;
	// EN: Sheet stack discharge conveyor speed reference [m/min].
	// PT: Referência de velocidade da esteira de descarga da pilha [m/min].
	sheetStackDischargeConveyorSpeedRefMPM  : REAL;

    //==============================================================
    // Backstop speed reference output
    //==============================================================
    // EN: Backstop speed reference [mm/s], always positive.
    // PT: Referência de velocidade do backstop [mm/s], sempre positiva.
    backstopSpeedRefMmps                : REAL;
	
	
	
    backstopPlateUpSolenoid                : BOOL;


    //==============================================================
    // Backstop encoder set outputs
    //==============================================================
    // EN: Pulse output to set/reset backstop encoder position.
    // PT: Pulso de saída para setar/resetar a posição do encoder do backstop.
    backstopSetEncoderPosition          : BOOL;

    // EN: Position value to set in the encoder block [mm].
    // PT: Valor de posição a ser gravado no bloco do encoder [mm].
    backstopSetEncoderPositionMm        : REAL;


    //==============================================================
    // Pneumatic valve outputs
    //==============================================================
    brakeValve                          : BOOL;

    sheetBrush1Valve                    : BOOL;
    sheetBrush2Valve                    : BOOL;
    sheetBrush3Valve                    : BOOL;

    brakeBrushValve                     : BOOL;
    backstopUpValve                     : BOOL;
    noCrushRollersUpDownValve               : BOOL;

	// EN: Sheet stack alignment brush output.
	//     TRUE = lowered/engaged; FALSE = raised/disengaged.
	// PT: Saída da vassoura de alinhamento da pilha de chapas.
	//     TRUE = abaixada/acionada; FALSE = levantada/desacionada.
	sheetStackAlignmentBrush              : BOOL;


    //==============================================================
    // General status outputs
    //==============================================================
    deviceState                         : STRING(30);

    faultActive                         : BOOL;
    synchronizedConveyorsRunning        : BOOL;


    //==============================================================
    // Sheet stack separation status outputs
    //==============================================================
    sheetStackSeparationState           : STRING(30);
    sheetStackSeparationStateCode       : INT;

    sheetStackSeparationReady           : BOOL;
    sheetStackSeparationActive          : BOOL;

    // EN: One-scan pulse when sheet stack separation starts.
    // PT: Pulso de um ciclo quando inicia a separação da pilha de chapas.
    sheetStackSeparationStarted         : BOOL;

    // EN: One-scan pulse when sheet stack separation finishes.
    // PT: Pulso de um ciclo quando finaliza a separação da pilha de chapas.
    sheetStackSeparationFinished        : BOOL;

    // EN: Brake active during sheet stack separation.
    // PT: Freio ativo durante a separação da pilha de chapas.
    sheetStackBrakeActive               : BOOL;


    //==============================================================
    // Sheet conveyor 2 separation status outputs
    //==============================================================
    sheetConveyor2SeparationActive      : BOOL;

    // EN: One-scan pulse when conveyor 2 separation tracking starts.
    // PT: Pulso de um ciclo quando inicia o rastreamento de separação da esteira 2.
    sheetConveyor2SeparationStarted     : BOOL;

    // EN: One-scan pulse when conveyor 2 separation tracking finishes.
    // PT: Pulso de um ciclo quando finaliza o rastreamento de separação da esteira 2.
    sheetConveyor2SeparationFinished    : BOOL;

    sheetConveyor2HighSpeedActive       : BOOL;

    // EN: Current conveyor 2 separation tracking distance [m].
    // PT: Distância atual rastreada na separação da esteira 2 [m].
    sheetConveyor2TrackingDistanceM     : REAL;

    // EN: Conveyor 2 separation target distance [m].
    // PT: Distância alvo de separação da esteira 2 [m].
    sheetConveyor2TargetDistanceM       : REAL;


    //==============================================================
    // Sheet conveyor 3 separation status outputs
    //==============================================================
    sheetConveyor3SeparationActive      : BOOL;

    // EN: One-scan pulse when conveyor 3 separation tracking starts.
    // PT: Pulso de um ciclo quando inicia o rastreamento de separação da esteira 3.
    sheetConveyor3SeparationStarted     : BOOL;

    // EN: One-scan pulse when conveyor 3 separation tracking finishes.
    // PT: Pulso de um ciclo quando finaliza o rastreamento de separação da esteira 3.
    sheetConveyor3SeparationFinished    : BOOL;

    sheetConveyor3HighSpeedActive       : BOOL;

    // EN: Current conveyor 3 separation tracking distance [m].
    // PT: Distância atual rastreada na separação da esteira 3 [m].
    sheetConveyor3TrackingDistanceM     : REAL;

    // EN: Conveyor 3 separation target distance [m].
    // PT: Distância alvo de separação da esteira 3 [m].
    sheetConveyor3TargetDistanceM       : REAL;

	//==============================================================
	// Conveyor leveler encoder set outputs
	//==============================================================
	// EN: Pulse output to set/reset conveyor leveler encoder position.
	// PT: Pulso de saída para setar/resetar a posição do encoder do nivelador.
	conveyorLevelerSetEncoderPosition   : BOOL;
	
	// EN: Position value to set in the conveyor leveler encoder block [mm].
	// PT: Valor de posição a ser gravado no bloco do encoder do nivelador [mm].
	conveyorLevelerSetEncoderPositionMm : REAL;
	
	
	//==============================================================
	// Conveyor leveler status outputs
	//==============================================================
	conveyorLevelerState                : STRING(30);
	
	conveyorLevelerHomed                : BOOL;
	conveyorLevelerInPosition           : BOOL;
	conveyorLevelerFault                : BOOL;
	conveyorLevelerFaultCode            : INT;
	
	// EN: Current calculated conveyor leveler target position [mm].
	// PT: Posição alvo calculada atual do nivelador [mm].
	conveyorLevelerTargetPositionMm     : REAL;
	
	// EN: Current conveyor leveler position error [mm].
	// PT: Erro atual de posição do nivelador [mm].
	conveyorLevelerPositionErrorMm      : REAL;

    //==============================================================
    // Backstop status outputs
    //==============================================================
    backstopState                       : STRING(30);

    backstopHomed                       : BOOL;
    backstopInPosition                  : BOOL;
    backstopFault                       : BOOL;
    backstopFaultCode                   : INT;

    // EN: Current calculated target position [mm].
    // PT: Posição alvo calculada atualmente [mm].
    backstopTargetPositionMm            : REAL;

    // EN: Current position error [mm].
    // PT: Erro atual de posição [mm].
    backstopPositionErrorMm             : REAL;
	
	//==============================================================
	// Sheet stack discharge conveyor control state
	//==============================================================
	sheetStackDischargeConveyorState               : STRING(30);
	sheetStackDischargeConveyorFault               : BOOL;
	sheetStackDischargeConveyorFaultCode           : INT;
	
	//==============================================================
	// Sheet stack discharge sequence status outputs
	//==============================================================
	sheetStackDischargeState                : STRING(30);
	sheetStackDischargeStateCode            : INT;
	
	sheetStackDischargePending              : BOOL;
	sheetStackDischargeActive               : BOOL;
	sheetStackDischargeStarted              : BOOL;
	sheetStackDischargeFinished             : BOOL;
	
	sheetStackDischargeFault                : BOOL;
	sheetStackDischargeFaultCode            : INT;
	
	//==============================================================
	// Sheet stack discharge last cycle diagnostic outputs
	//==============================================================
	sheetStackDischargeLastCycleOk          : BOOL;
	sheetStackDischargeLastResultCode       : INT;
	sheetStackDischargeLastFaultStepCode    : INT;
	sheetStackDischargeLastFaultCode        : INT;	

END_VAR

VAR
	
	//==============================================================
	// Stop machine pulse control
	//==============================================================
	stopMachineFaultCondition     : BOOL;
	stopMachineFaultConditionOld  : BOOL;
	rStopMachineFaultCondition    : BOOL;
	
	tpStopMachinePulse            : TP;
	
	//==============================================================
	// Backstop manual intervention memory
	//==============================================================
	backstopManualInterventionActive     : BOOL;
	backstopManualInterventionPositionMm : REAL;
	
	//==============================================================
	// Sheet stack discharge backstop latched targets
	//==============================================================
	backstopProgrammedDischargeTargetMm : REAL;
	backstopDischargeOpenBasePositionMm : REAL;
	backstopDischargeOpenTargetMm       : REAL;
	
	//==============================================================
	// Backstop automatic positioning command control
	//==============================================================
	backstopExecutePositioningCmdOld    : BOOL;
	rBackstopExecutePositioning         : BOOL;
	
	backstopTargetOverrideOld           : BOOL;
	backstopTargetOverrideFallingEdge   : BOOL;
	
	backstopPositioningRequestActive    : BOOL;
	backstopLatchedTargetPositionMm     : REAL;
	backstopProgrammedTargetPositionMm  : REAL;
	
	//==============================================================
	// Backstop manual intervention memory
	//==============================================================
	// EN: Used by automatic discharge sequence to avoid closing onto material
	//     after operator manual intervention.

	//==============================================================
	// Backstop encoder set pulse
	//==============================================================
	backstopSetEncoderPositionTrigger  : BOOL;
	tpBackstopSetEncoderPosition       : TP;

	//==============================================================
	// Sheet stack discharge backstop latched targets
	//==============================================================

    //==============================================================
    // Group state machine
    //==============================================================
    syncConveyorsState                  : INT;


    //==============================================================
    // Package separation state machine
    //==============================================================
    packageSeparationState              : INT;


    //==============================================================
    // Backstop state machine
    //==============================================================
    backstopControlState                : INT;


    //==============================================================
    // Edge detection
    //==============================================================
    startCmdOld                         : BOOL;
    stopCmdOld                          : BOOL;
    stackerUnloadCmdOld                  : BOOL;
    changeBatchCmdOld                    : BOOL;

    backstopHomeCmdOld                  : BOOL;


    //==============================================================
    // Internal conditions
    //==============================================================
    allSynchronizedDrivesOk             : BOOL;
    anyFault                            : BOOL;
    speedControlEnabled                 : BOOL;
    rampReset                           : BOOL;


    //==============================================================
    // Sheet length conversion
    //==============================================================
    // EN: Internal sheet length converted from mm to m.
    // PT: Comprimento interno da chapa convertido de mm para m.
    sheetLengthM                        : REAL;


    //==============================================================
    // Normal speed calculation
    //==============================================================
    effectiveLineSpeedMPM                : REAL;
    normalStackerSpeedMPM               : REAL;

    sheetConveyor1NormalSpeedMPM        : REAL;
    sheetConveyor2NormalSpeedMPM        : REAL;
    sheetConveyor3NormalSpeedMPM        : REAL;
    conveyorLevelerNormalSpeedMPM       : REAL;


    //==============================================================
    // Package gap speed calculation
    //==============================================================
    sheetConveyor1GapSpeedMPM           : REAL;
    sheetConveyor2GapSpeedMPM           : REAL;
    sheetConveyor3GapSpeedMPM           : REAL;


    //==============================================================
    // Speed targets
    //==============================================================
    sheetConveyor1TargetSpeedMPM        : REAL;
    sheetConveyor2TargetSpeedMPM        : REAL;
    sheetConveyor3TargetSpeedMPM        : REAL;
    conveyorLevelerTargetSpeedMPM       : REAL;


    //==============================================================
    // Package gap distance calculation
    //==============================================================
    packageGapDistanceTargetM           : REAL;

    sheetConveyor2OpeningSpeedMPM       : REAL;
    sheetConveyor3OpeningSpeedMPM       : REAL;

    sheetConveyor2OpeningDistanceM      : REAL;
    sheetConveyor3OpeningDistanceM      : REAL;


	//==============================================================
	// Conveyor leveler state machine
	//==============================================================
	conveyorLevelerControlState         : INT;
	
	
	//==============================================================
	// Conveyor leveler edge detection
	//==============================================================
	conveyorLevelerHomeCmdOld           : BOOL;
	rConveyorLevelerHome                : BOOL;
	
	
	//==============================================================
	// Conveyor leveler encoder set pulse
	//==============================================================
	conveyorLevelerSetEncoderPositionTrigger   : BOOL;
	tpConveyorLevelerSetEncoderPosition        : TP;
	
	
	//==============================================================
	// Conveyor leveler control calculation
	//==============================================================
	conveyorLevelerAutoTargetPositionMm        : REAL;
	conveyorLevelerRawSpeedRefMmps             : REAL;
	
	// EN: Internal signed speed command. Positive = up, negative = down.
	// PT: Comando interno de velocidade com sinal. Positivo = subir, negativo = descer.
	conveyorLevelerSignedSpeedRefMmps          : REAL;
	
	conveyorLevelerAbsPositionErrorMm          : REAL;
	
	
	//==============================================================
	// Conveyor leveler movement permissions
	//==============================================================
	conveyorLevelerUpAllowed                   : BOOL;
	conveyorLevelerDownAllowed                 : BOOL;
	
	conveyorLevelerMoveRequest                 : BOOL;
	conveyorLevelerBrakeReleaseRequest         : BOOL;
	
	
	//==============================================================
	// Conveyor leveler homing
	//==============================================================
	conveyorLevelerHomeLimitReached            : BOOL;
	conveyorLevelerHomeMoveAllowed             : BOOL;
	
	
	//==============================================================
	// Conveyor leveler timers
	//==============================================================
	tonConveyorLevelerHomingTimeout            : TON;
	
	// EN: Delay after brake release before motor movement.
	// PT: Atraso após liberar o freio antes de movimentar o motor.
	tonConveyorLevelerBrakeReleaseDelay        : TON;
	
	// EN: Keeps brake released for a short time after movement stops.
	// PT: Mantém o freio liberado por um tempo após parar o movimento.
	tonConveyorLevelerBrakeHoldDelay           : TON;
	
	
	//==============================================================
	// Conveyor leveler speed ramp instance
	//==============================================================
	// EN: Ramp used for conveyor leveler vertical speed [mm/s].
	// PT: Rampa usada para velocidade vertical do nivelador [mm/s].
	instRampConveyorLeveler                    : FB_Gen_SRamp;
	

    //==============================================================
    // Backstop control calculation
    //==============================================================
    backstopAutoTargetPositionMm        : REAL;
    backstopRawSpeedRefMmps             : REAL;
    backstopAbsPositionErrorMm          : REAL;

    backstopHomeLimitReached            : BOOL;
    backstopOpenAllowed                 : BOOL;
    backstopCloseAllowed                : BOOL;

    rBackstopHome                       : BOOL;


	//==============================================================
	// Backstop homing edge detection
	//==============================================================
	backstopHomeLimitOld                 : BOOL;
	backstopHomeLimitFallingEdge         : BOOL;
	backstopHomeMoveAllowed              : BOOL;
	
	
	
	//==============================================================
	// Backstop timers
	//==============================================================
	tonBackstopHomeSettleDelay           : TON;



    //==============================================================
    // Backstop timers
    //==============================================================
    tonBackstopHomingTimeout            : TON;


    //==============================================================
    // Speed ramp instances
    //==============================================================
    instRampSheetConveyor1              : FB_Gen_SRamp;
    instRampSheetConveyor2              : FB_Gen_SRamp;
    instRampSheetConveyor3              : FB_Gen_SRamp;


    //==============================================================
    // PLC scan time measurement
    //==============================================================
    instCycleTime                       : CYCLE_TIME;
    scanTimeS                           : REAL;
    scanTimeMs                          : REAL;

	backstopSignedSpeedRefMmps: REAL;
	
	//==============================================================
	// Sheet stack discharge state machine
	//==============================================================
	sheetStackDischargeControlState         : INT;

	// EN: Keeps the alignment brush raised throughout the discharge cycle.
	// PT: Mantém a vassoura de alinhamento levantada durante todo o descarte.
	sheetStackAlignmentBrushLiftedForDischarge : BOOL;
	
	
	//==============================================================
	// Sheet stack discharge request control
	//==============================================================
	// EN: Prevents a maintained automatic request from being accepted
	//     more than once before packageCompleteCmd returns to FALSE.
	// PT: Impede que uma solicitação automática mantida seja aceita mais
	//     de uma vez antes de packageCompleteCmd retornar para FALSE.
	packageCompleteCmdAccepted              : BOOL;
	changeBatchRequestPending               : BOOL;
	changeBatchCycleActive                  : BOOL;

	// EN: Internal one-scan event generated for any accepted unload source.
	// PT: Evento interno de um scan gerado para qualquer fonte de descarte aceita.
	dischargeRequestAccepted                : BOOL;

	tpExternalCounterReset                  : TP;
	
	
	//==============================================================
	// Sheet stack discharge timers
	//==============================================================
	tonSheetStackDischarge                  : TON;
	
	
	//==============================================================
	// Sheet stack discharge internal conditions
	//==============================================================
	sheetStackDischargeFaultCondition       : BOOL;
	
	
	//==============================================================
	// Backstop target override
	//==============================================================
	backstopTargetOverrideActive            : BOOL;
	backstopTargetOverridePositionMm        : REAL;
	
	
	//==============================================================
	// Conveyor leveler target override
	//==============================================================
	conveyorLevelerTargetOverrideActive     : BOOL;
	conveyorLevelerTargetOverridePositionMm : REAL;	
	
	
	sheetStackDischargeConveyorRunRequest: BOOL;
	instTONBackstopDownDelay: TON;
	
	//==============================================================
	// Sheet stack discharge step timeout
	//==============================================================
	tonSheetStackDischargeStepTimeout       : TON;
	
	sheetStackDischargeCycleHasManualSkip   : BOOL;
	sheetStackDischargeCycleHasTimeout      : BOOL;	
	
	
	//==============================================================
	// Conveyor leveler homing edge detection
	//==============================================================
	conveyorLevelerHomeLimitOld                 : BOOL;
	conveyorLevelerHomeLimitFallingEdge         : BOOL;	

	//==============================================================
	// System master run control
	//==============================================================
	systemRunEnable : BOOL;
	
	rStartCmd : BOOL;
	rStopCmd  : BOOL;
	
	//==============================================================
	// Automatic homing requests generated by master start
	//==============================================================
	backstopAutoHomeRequest        : BOOL;
	conveyorLevelerAutoHomeRequest : BOOL;

	// EN: Latched start requests awaiting valid homing permissives.
	// PT: Pedidos de partida memorizados aguardando permissivos válidos de homing.
	backstopAutoHomePending        : BOOL;
	conveyorLevelerAutoHomePending : BOOL;
	
	//==============================================================
	// Conveyor leveler home request command control
	//==============================================================
	conveyorLevelerHomeRequestCombined    : BOOL;
	conveyorLevelerHomeRequestCombinedOld : BOOL;
	backstopHomeRunning: BOOL;
	//==============================================================
	// Backstop home request command control
	//==============================================================
	backstopHomeRequestCombined    : BOOL;
	backstopHomeRequestCombinedOld : BOOL;
	
	

END_VAR

_SystemControl();

_SheetConveyorGroupControl();
_ConveyorSpeedControl();
_SheetStackDischargeControl();

_BackstopControl();
_ConveyorLevelerControl();
_SheetStackAlignmentBrushControl();
_SheetStackDischargeConveyorControl();
_MachineAuxiliary();
_HmiStatus();
_AlarmControl();

//==============================================================
// SIMPLE STACKER — ALARM CONTROL
// EN: Maps internal faults and status conditions to HMI alarm structure.
//==============================================================
METHOD _AlarmControl

VAR
	hmiAlarmsNotActive: hmiAlarmsSimpleStacker_TypeStruct;
END_VAR
//==============================================================
// HMI alarms reset / latch logic
//==============================================================

IF resetCmd THEN

    // Reset geral dos alarmes
    hmiAlarms := hmiAlarmsNotActive;

ELSE

    //==============================================================
    // 1) General / system alarms
    //==============================================================
    hmiAlarms.safetyCircuitNotOk :=
        hmiAlarms.safetyCircuitNotOk OR
        NOT safetyCircuitOk;

    hmiAlarms.systemFaultActive :=
        hmiAlarms.systemFaultActive OR
        faultActive OR
        backstopFault OR
        conveyorLevelerFault OR
        sheetStackDischargeFault OR
        sheetStackDischargeConveyorFault;

    hmiAlarms.systemNotEnabled :=
        hmiAlarms.systemNotEnabled OR
        NOT systemRunEnable;

    // EN: These generic safety feedbacks are used only for diagnostics.
    // PT: Estes retornos genéricos de segurança são usados apenas para diagnóstico.
    hmiAlarms.safetyFeedback1NotOk := NOT safetyFeedBack1;
    hmiAlarms.safetyFeedback2NotOk := NOT safetyFeedBack2;
    hmiAlarms.safetyFeedback3NotOk := NOT safetyFeedBack3;
    hmiAlarms.safetyFeedback4NotOk := NOT safetyFeedBack4;
    hmiAlarms.safetyFeedback5NotOk := NOT safetyFeedBack5;
    hmiAlarms.safetyFeedback6NotOk := NOT safetyFeedBack6;
    hmiAlarms.safetyFeedback7NotOk := NOT safetyFeedBack7;
    hmiAlarms.safetyFeedback8NotOk := NOT safetyFeedBack8;


    //==============================================================
    // 2) Sheet conveyor group alarms
    //==============================================================
    hmiAlarms.sheetConveyor1DriveNotOk :=
        hmiAlarms.sheetConveyor1DriveNotOk OR
        NOT sheetConveyor1DriveOk;

    hmiAlarms.sheetConveyor2DriveNotOk :=
        hmiAlarms.sheetConveyor2DriveNotOk OR
        NOT sheetConveyor2DriveOk;

    hmiAlarms.sheetConveyor3DriveNotOk :=
        hmiAlarms.sheetConveyor3DriveNotOk OR
        NOT sheetConveyor3DriveOk;

    hmiAlarms.sheetConveyorGroupFault :=
        hmiAlarms.sheetConveyorGroupFault OR
        NOT safetyCircuitOk OR
        NOT sheetConveyor1DriveOk OR
        NOT sheetConveyor2DriveOk OR
        NOT sheetConveyor3DriveOk;

 //   hmiAlarms.synchronizedConveyorsNotRunning :=
 //       hmiAlarms.synchronizedConveyorsNotRunning OR
 //       (
 //           systemRunEnable AND
 //           NOT synchronizedConveyorsRunning
 //       );


    //==============================================================
    // 3) Sheet stack separation alarms / indications
    //==============================================================
    // Mantido comentado conforme lógica original.
    // Se quiser ativar como latch, use o mesmo padrão:
    //
    // hmiAlarms.sheetStackSeparationNotReady :=
    //     hmiAlarms.sheetStackSeparationNotReady OR
    //     (
    //         systemRunEnable AND
    //         synchronizedConveyorsRunning AND
    //         NOT sheetStackSeparationReady
    //     );
    //
    // hmiAlarms.sheetStackSeparationActive :=
    //     hmiAlarms.sheetStackSeparationActive OR
    //     sheetStackSeparationActive;
    //
    // hmiAlarms.sheetStackBrakeActive :=
    //     hmiAlarms.sheetStackBrakeActive OR
    //     sheetStackBrakeActive;


    //==============================================================
    // 4) Sheet stack discharge sequence alarms / indications
    //==============================================================
    hmiAlarms.sheetStackDischargeFault :=
        hmiAlarms.sheetStackDischargeFault OR
        sheetStackDischargeFault;

    hmiAlarms.sheetStackDischargeLastCycleNotOk :=
        hmiAlarms.sheetStackDischargeLastCycleNotOk OR
        (
            NOT sheetStackDischargeLastCycleOk AND
            sheetStackDischargeLastResultCode <> 0
        );

    hmiAlarms.sheetStackDischargeTimeout :=
        hmiAlarms.sheetStackDischargeTimeout OR
        sheetStackDischargeLastResultCode = 3;

    hmiAlarms.sheetStackDischargeManualSkip :=
        hmiAlarms.sheetStackDischargeManualSkip OR
        sheetStackDischargeLastResultCode = 2;


    //==============================================================
    // 5) Sheet stack discharge conveyor alarms
    //==============================================================
    hmiAlarms.sheetStackDischargeConveyorDriveNotOk :=
        hmiAlarms.sheetStackDischargeConveyorDriveNotOk OR
        NOT sheetStackDischargeConveyorDriveOk;

    hmiAlarms.sheetStackDischargeConveyorFault :=
        hmiAlarms.sheetStackDischargeConveyorFault OR
        sheetStackDischargeConveyorFault;


    //==============================================================
    // 6) Backstop alarms / indications
    //==============================================================
    hmiAlarms.backstopDriveNotOk :=
        hmiAlarms.backstopDriveNotOk OR
        NOT backstopDriveOk;

    hmiAlarms.backstopFault :=
        hmiAlarms.backstopFault OR
        backstopFault;

    hmiAlarms.backstopNotHomed :=
        hmiAlarms.backstopNotHomed OR
        (
            backstopAutoCmd AND
            NOT backstopHomed
        );

    (*
    hmiAlarms.backstopNotInPosition :=
        hmiAlarms.backstopNotInPosition OR
        (
            systemRunEnable AND
            backstopAutoCmd AND
            backstopHomed AND
            NOT backstopInPosition AND
            NOT backstopTargetOverrideActive
        );
    *)

    hmiAlarms.backstopSafeMaxLimitActive :=
        hmiAlarms.backstopSafeMaxLimitActive OR
        backstopSafeMaxLimit;

    hmiAlarms.backstopSafeMinLimitActive :=
        hmiAlarms.backstopSafeMinLimitActive OR
        backstopSafeMinLimit;

